      A     M      3.3;
      =     L      0.0;
      A     L      0.0;
      A     I     45.0;
      AN    I     45.1;
      =     M    612.2;
      A     L      0.0;
      AN    I     45.0;
      A     I     45.1;
      =     M    612.3;
NETWORK
TITLE =GUN3 1ST SHIFT ADV/REV END (LH ONLY)

      A     M      3.3;
      =     L      0.0;
      A     L      0.0;
      A     I     45.2;
      AN    I     45.3;
      =     M    612.4;
      A     L      0.0;
      AN    I     45.2;
      A     I     45.3;
      =     M    612.5;
NETWORK
TITLE =GUN3 2ND SHIFT ADV/REV END (LH ONLY)

      A     M      3.3;
      =     L      0.0;
      A     L      0.0;
      A     I     45.4;
      AN    I     45.5;
      =     M    612.6;
      A     L      0.0;
      AN    I     45.4;
      A     I     45.5;
      =     M    612.7;
NETWORK
TITLE =ALL CLAMP ADV/REV END

      A     M      3.3;
      =     L      0.0;
      A     L      0.0;
      A     M    610.2;
      A     M    610.4;
      =     M    618.0;
      A     L      0.0;
      A     M    610.3;
      A     M    610.5;
      =     M    618.1;
NETWORK
TITLE =GUN ALL HOME POSI.
//G3 SHIFT= LH ONLY
      A     M    612.1;
      A     M    612.2;
      A     M    612.5;
      A     M    612.7;
      =     M    618.2;
NETWORK
TITLE =PIN ADV
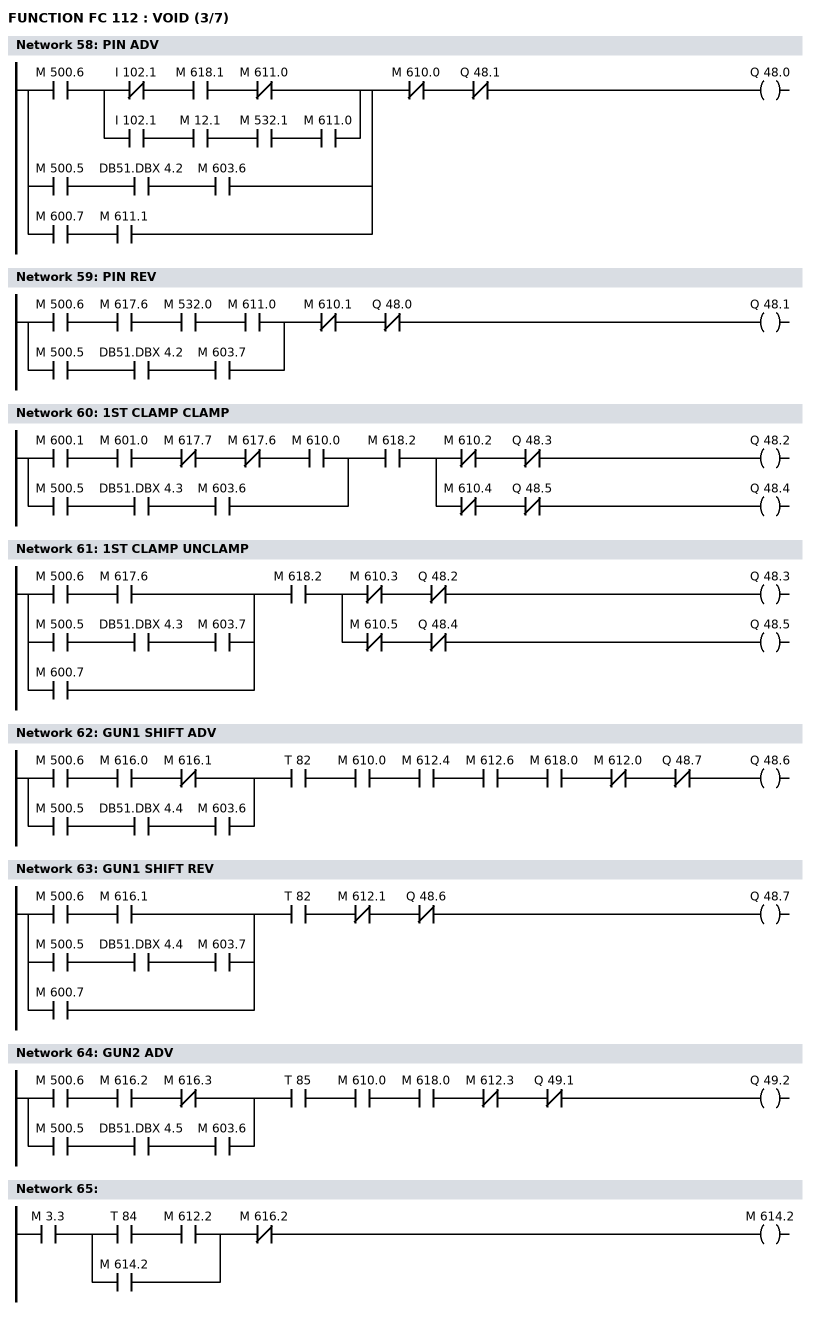

      A(    ;
      A     M    500.6;
      A(    ;
      AN    I    102.1;
      A     M    618.1;
      AN    M    611.0;
      O     ;
      A     I    102.1;
      A     M     12.1;
      A     M    532.1;
      A     M    611.0;
      )     ;
      O     ;
      A     M    500.5;
      A     DB51.DBX    4.2;
      A     M    603.6;
      O     ;
      A     M    600.7;
      A     M    611.1;
      )     ;
      AN    M    610.0;
      AN    Q     48.1;
      =     Q     48.0;
NETWORK
TITLE =PIN REV

      A(    ;
      A     M    500.6;
      A     M    617.6;
      A     M    532.0;
      A     M    611.0;
      O     ;
      A     M    500.5;
      A     DB51.DBX    4.2;
      A     M    603.7;
      )     ;
      AN    M    610.1;
      AN    Q     48.0;
      =     Q     48.1;
NETWORK
TITLE =1ST CLAMP CLAMP

      A(    ;
      A     M    600.1;
      A     M    601.0;
      AN    M    617.7;
      AN    M    617.6;
      A     M    610.0;
      O     ;
      A     M    500.5;
      A     DB51.DBX    4.3;
      A     M    603.6;
      )     ;
      A     M    618.2;
      =     L      0.0;
      A     L      0.0;
      AN    M    610.2;
      AN    Q     48.3;
      =     Q     48.2;
      A     L      0.0;
      AN    M    610.4;
      AN    Q     48.5;
      =     Q     48.4;
NETWORK
TITLE =1ST CLAMP UNCLAMP

      A(    ;
      A     M    500.6;
      A     M    617.6;
      O     ;
      A     M    500.5;
      A     DB51.DBX    4.3;
      A     M    603.7;
      O     M    600.7;
      )     ;
      A     M    618.2;
      =     L      0.0;
      A     L      0.0;
      AN    M    610.3;
      AN    Q     48.2;
      =     Q     48.3;
      A     L      0.0;
      AN    M    610.5;
      AN    Q     48.4;
      =     Q     48.5;
NETWORK
TITLE =GUN1 SHIFT ADV

      A(    ;
      A     M    500.6;
      A     M    616.0;
      AN    M    616.1;
      O     ;
      A     M    500.5;
      A     DB51.DBX    4.4;
      A     M    603.6;
      )     ;
      A     T     82;
      A     M    610.0;
      A     M    612.4;
      A     M    612.6;
      A     M    618.0;
      AN    M    612.0;
      AN    Q     48.7;
      =     Q     48.6;
NETWORK
TITLE =GUN1 SHIFT REV

      A(    ;
      A     M    500.6;
      A     M    616.1;
      O     ;
      A     M    500.5;
      A     DB51.DBX    4.4;
      A     M    603.7;
      O     M    600.7;
      )     ;
      A     T     82;
      AN    M    612.1;
      AN    Q     48.6;
      =     Q     48.7;
NETWORK
TITLE =GUN2 ADV

      A(    ;
      A     M    500.6;
      A     M    616.2;
      AN    M    616.3;
      O     ;
      A     M    500.5;
      A     DB51.DBX    4.5;
      A     M    603.6;
      )     ;
      A     T     85;
      A     M    610.0;
      A     M    618.0;
      AN    M    612.3;
      AN    Q     49.1;
      =     Q     49.2;
NETWORK
TITLE =

      A     M      3.3;
      A(    ;
      A     T     84;
      A     M    612.2;
      O     M    614.2;
      )     ;
      AN    M    616.2;
      =     M    614.2;
NETWORK
TITLE =GUN2 REV
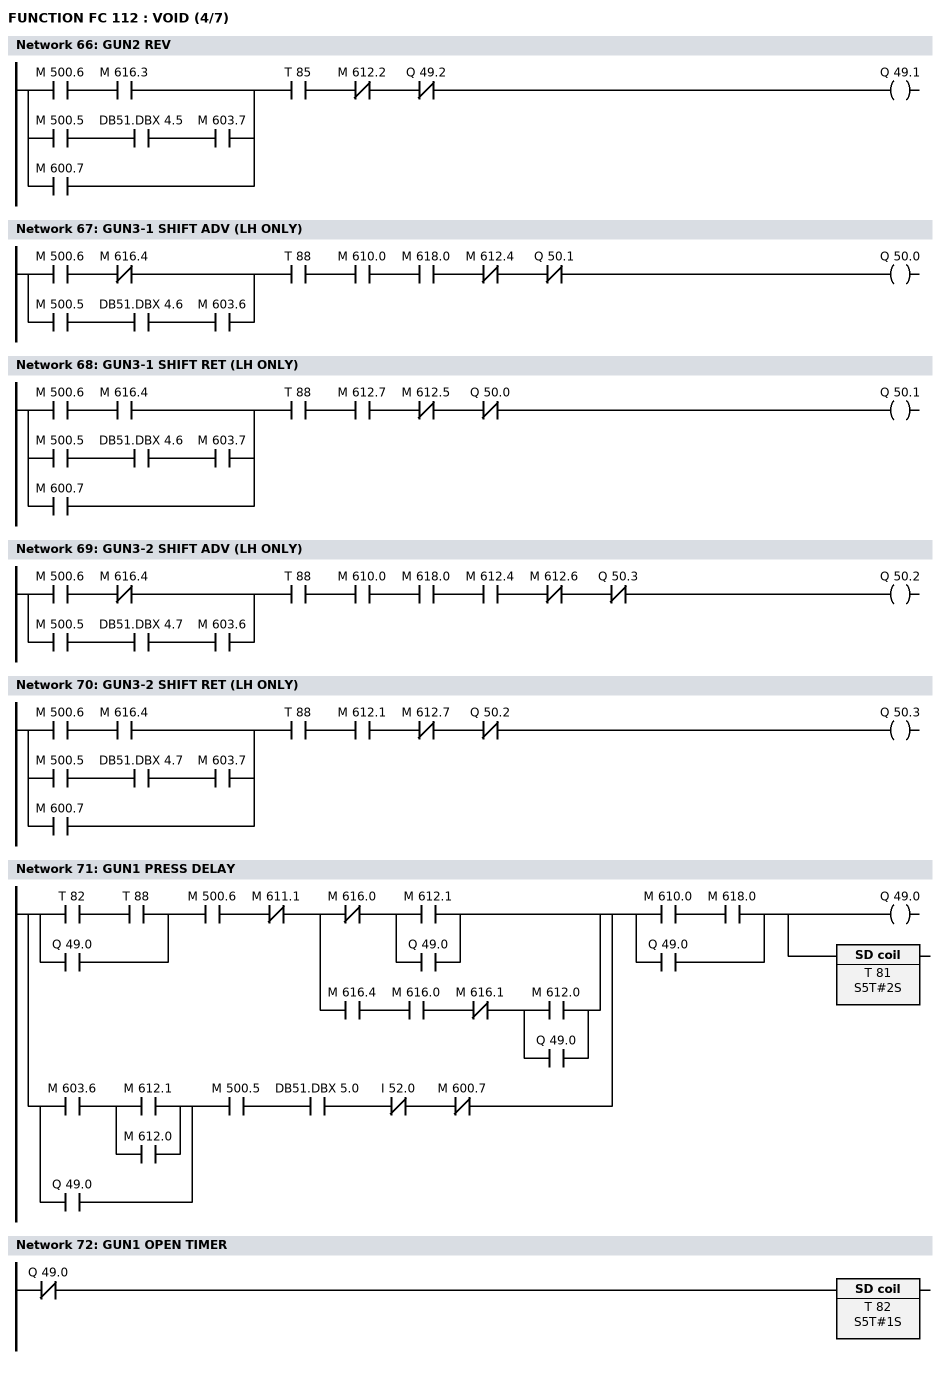

      A(    ;
      A     M    500.6;
      A     M    616.3;
      O     ;
      A     M    500.5;
      A     DB51.DBX    4.5;
      A     M    603.7;
      O     M    600.7;
      )     ;
      A     T     85;
      AN    M    612.2;
      AN    Q     49.2;
      =     Q     49.1;
NETWORK
TITLE =GUN3-1 SHIFT ADV (LH ONLY)

      A(    ;
      A     M    500.6;
      AN    M    616.4;
      O     ;
      A     M    500.5;
      A     DB51.DBX    4.6;
      A     M    603.6;
      )     ;
      A     T     88;
      A     M    610.0;
      A     M    618.0;
      AN    M    612.4;
      AN    Q     50.1;
      =     Q     50.0;
NETWORK
TITLE =GUN3-1 SHIFT RET (LH ONLY)

      A(    ;
      A     M    500.6;
      A     M    616.4;
      O     ;
      A     M    500.5;
      A     DB51.DBX    4.6;
      A     M    603.7;
      O     M    600.7;
      )     ;
      A     T     88;
      A     M    612.7;
      AN    M    612.5;
      AN    Q     50.0;
      =     Q     50.1;
NETWORK
TITLE =GUN3-2 SHIFT ADV (LH ONLY)

      A(    ;
      A     M    500.6;
      AN    M    616.4;
      O     ;
      A     M    500.5;
      A     DB51.DBX    4.7;
      A     M    603.6;
      )     ;
      A     T     88;
      A     M    610.0;
      A     M    618.0;
      A     M    612.4;
      AN    M    612.6;
      AN    Q     50.3;
      =     Q     50.2;
NETWORK
TITLE =GUN3-2 SHIFT RET (LH ONLY)

      A(    ;
      A     M    500.6;
      A     M    616.4;
      O     ;
      A     M    500.5;
      A     DB51.DBX    4.7;
      A     M    603.7;
      O     M    600.7;
      )     ;
      A     T     88;
      A     M    612.1;
      AN    M    612.7;
      AN    Q     50.2;
      =     Q     50.3;
NETWORK
TITLE =GUN1 PRESS DELAY

      A(    ;
      A(    ;
      A     T     82;
      A     T     88;
      O     Q     49.0;
      )     ;
      A     M    500.6;
      AN    M    611.1;
      A(    ;
      AN    M    616.0;
      A(    ;
      O     M    612.1;
      O     Q     49.0;
      )     ;
      O     ;
      A     M    616.4;
      A     M    616.0;
      AN    M    616.1;
      A(    ;
      O     M    612.0;
      O     Q     49.0;
      )     ;
      )     ;
      O     ;
      A(    ;
      A     M    603.6;
      A(    ;
      O     M    612.1;
      O     M    612.0;
      )     ;
      O     Q     49.0;
      )     ;
      A     M    500.5;
      A     DB51.DBX    5.0;
      AN    I     52.0;
      AN    M    600.7;
      )     ;
      A(    ;
      A     M    610.0;
      A     M    618.0;
      O     Q     49.0;
      )     ;
      =     Q     49.0;
      L     S5T#2S;
      SD    T     81;
NETWORK
TITLE =GUN1 OPEN TIMER

      AN    Q     49.0;
      L     S5T#1S;
      SD    T     82;
NETWORK
TITLE =GUN2 PRESS DELAY
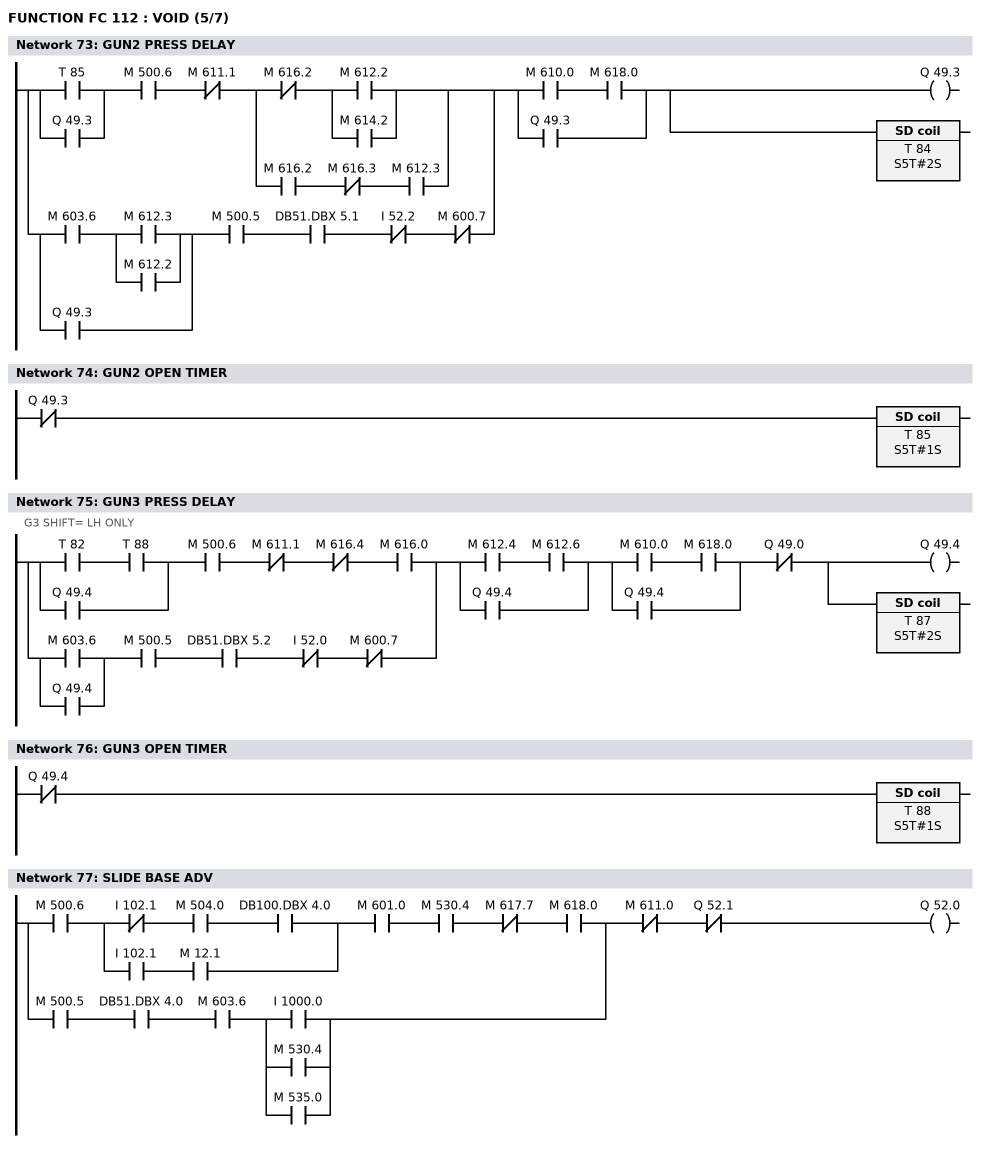

      A(    ;
      A(    ;
      O     T     85;
      O     Q     49.3;
      )     ;
      A     M    500.6;
      AN    M    611.1;
      A(    ;
      AN    M    616.2;
      A(    ;
      O     M    612.2;
      O     M    614.2;
      )     ;
      O     ;
      A     M    616.2;
      AN    M    616.3;
      A     M    612.3;
      )     ;
      O     ;
      A(    ;
      A     M    603.6;
      A(    ;
      O     M    612.3;
      O     M    612.2;
      )     ;
      O     Q     49.3;
      )     ;
      A     M    500.5;
      A     DB51.DBX    5.1;
      AN    I     52.2;
      AN    M    600.7;
      )     ;
      A(    ;
      A     M    610.0;
      A     M    618.0;
      O     Q     49.3;
      )     ;
      =     Q     49.3;
      L     S5T#2S;
      SD    T     84;
NETWORK
TITLE =GUN2 OPEN TIMER

      AN    Q     49.3;
      L     S5T#1S;
      SD    T     85;
NETWORK
TITLE =GUN3 PRESS DELAY
//G3 SHIFT= LH ONLY
      A(    ;
      A(    ;
      A     T     82;
      A     T     88;
      O     Q     49.4;
      )     ;
      A     M    500.6;
      AN    M    611.1;
      AN    M    616.4;
      A     M    616.0;
      O     ;
      A(    ;
      O     M    603.6;
      O     Q     49.4;
      )     ;
      A     M    500.5;
      A     DB51.DBX    5.2;
      AN    I     52.0;
      AN    M    600.7;
      )     ;
      A(    ;
      A     M    612.4;
      A     M    612.6;
      O     Q     49.4;
      )     ;
      A(    ;
      A     M    610.0;
      A     M    618.0;
      O     Q     49.4;
      )     ;
      AN    Q     49.0;
      =     Q     49.4;
      L     S5T#2S;
      SD    T     87;
NETWORK
TITLE =GUN3 OPEN TIMER

      AN    Q     49.4;
      L     S5T#1S;
      SD    T     88;
NETWORK
TITLE =SLIDE BASE ADV

      A(    ;
      A     M    500.6;
      A(    ;
      AN    I    102.1;
      A     M    504.0;
      A     DB100.DBX    4.0;
      O     ;
      A     I    102.1;
      A     M     12.1;
      )     ;
      A     M    601.0;
      A     M    530.4;
      AN    M    617.7;
      A     M    618.0;
      O     ;
      A     M    500.5;
      A     DB51.DBX    4.0;
      A     M    603.6;
      A(    ;
      O     I   1000.0;
      O     M    530.4;
      O     M    535.0;
      )     ;
      )     ;
      AN    M    611.0;
      AN    Q     52.1;
      =     Q     52.0;
NETWORK
TITLE =SLIDE BASE REV
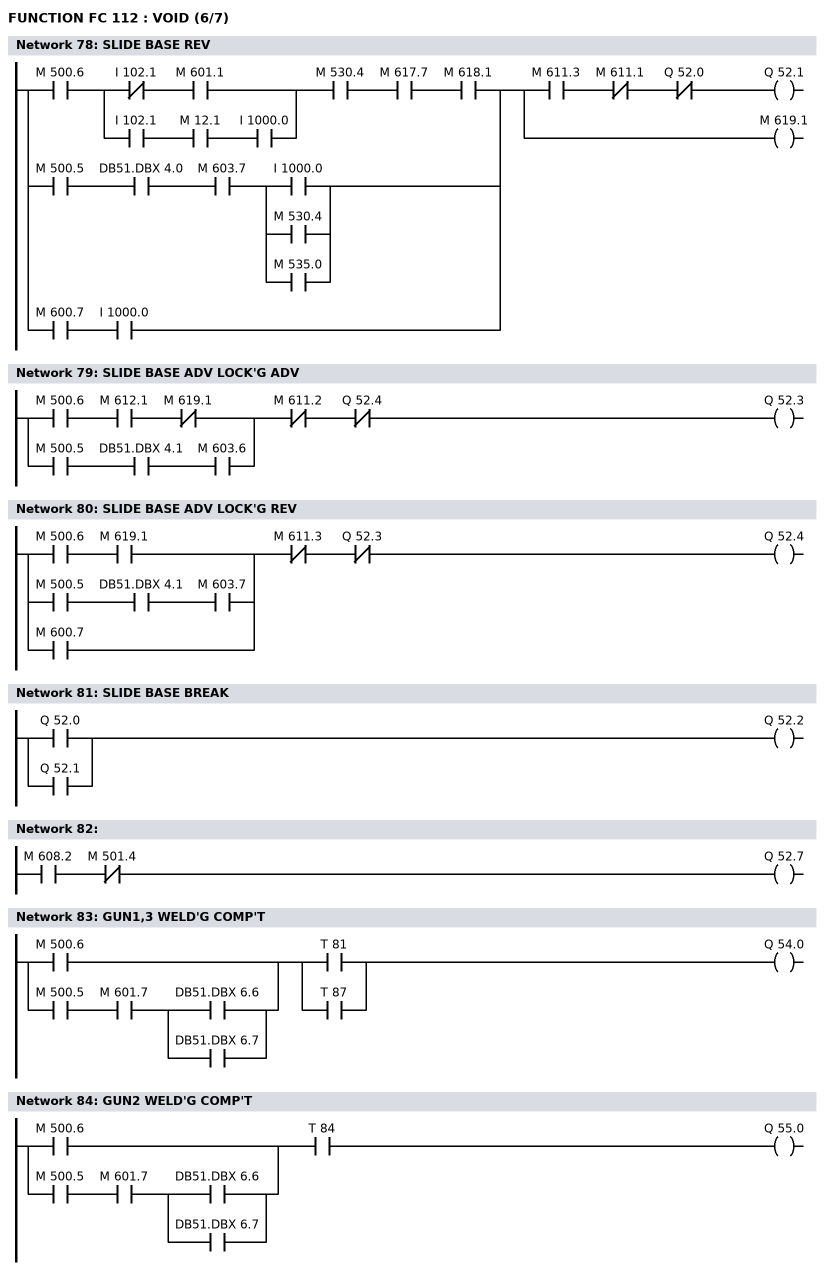

      A     M    500.6;
      A(    ;
      AN    I    102.1;
      A     M    601.1;
      O     ;
      A     I    102.1;
      A     M     12.1;
      A     I   1000.0;
      )     ;
      A     M    530.4;
      A     M    617.7;
      A     M    618.1;
      O     ;
      A     M    500.5;
      A     DB51.DBX    4.0;
      A     M    603.7;
      A(    ;
      O     I   1000.0;
      O     M    530.4;
      O     M    535.0;
      )     ;
      O     ;
      A     M    600.7;
      A     I   1000.0;
      =     L      0.0;
      A     L      0.0;
      A     M    611.3;
      AN    M    611.1;
      AN    Q     52.0;
      =     Q     52.1;
      A     L      0.0;
      BLD   102;
      =     M    619.1;
NETWORK
TITLE =SLIDE BASE ADV LOCK'G ADV

      A(    ;
      A     M    500.6;
      A     M    612.1;
      AN    M    619.1;
      O     ;
      A     M    500.5;
      A     DB51.DBX    4.1;
      A     M    603.6;
      )     ;
      AN    M    611.2;
      AN    Q     52.4;
      =     Q     52.3;
NETWORK
TITLE =SLIDE BASE ADV LOCK'G REV

      A(    ;
      A     M    500.6;
      A     M    619.1;
      O     ;
      A     M    500.5;
      A     DB51.DBX    4.1;
      A     M    603.7;
      O     M    600.7;
      )     ;
      AN    M    611.3;
      AN    Q     52.3;
      =     Q     52.4;
NETWORK
TITLE =SLIDE BASE BREAK

      O     Q     52.0;
      O     Q     52.1;
      =     Q     52.2;
NETWORK
TITLE =

      A     M    608.2;
      AN    M    501.4;
      =     Q     52.7;
NETWORK
TITLE =GUN1,3 WELD'G COMP'T

      A(    ;
      O     M    500.6;
      O     ;
      A     M    500.5;
      A     M    601.7;
      A(    ;
      O     DB51.DBX    6.6;
      O     DB51.DBX    6.7;
      )     ;
      )     ;
      A(    ;
      O     T     81;
      O     T     87;
      )     ;
      =     Q     54.0;
NETWORK
TITLE =GUN2 WELD'G COMP'T

      A(    ;
      O     M    500.6;
      O     ;
      A     M    500.5;
      A     M    601.7;
      A(    ;
      O     DB51.DBX    6.6;
      O     DB51.DBX    6.7;
      )     ;
      )     ;
      A     T     84;
      =     Q     55.0;
NETWORK
TITLE =GUN1,3 WELD'G TEST
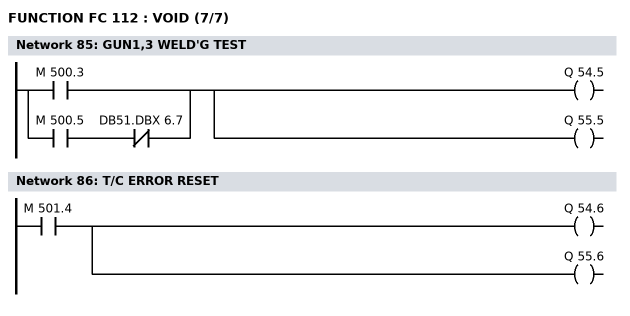

      O     M    500.3;
      O     ;
      A     M    500.5;
      AN    DB51.DBX    6.7;
      =     Q     54.5;
      =     Q     55.5;
NETWORK
TITLE =T/C ERROR RESET

      A     M    501.4;
      =     Q     54.6;
      =     Q     55.6;
END_FUNCTION

FUNCTION FC 113 : VOID
TITLE =
VERSION : 0.1

BEGIN
NETWORK
TITLE =BODY NO.
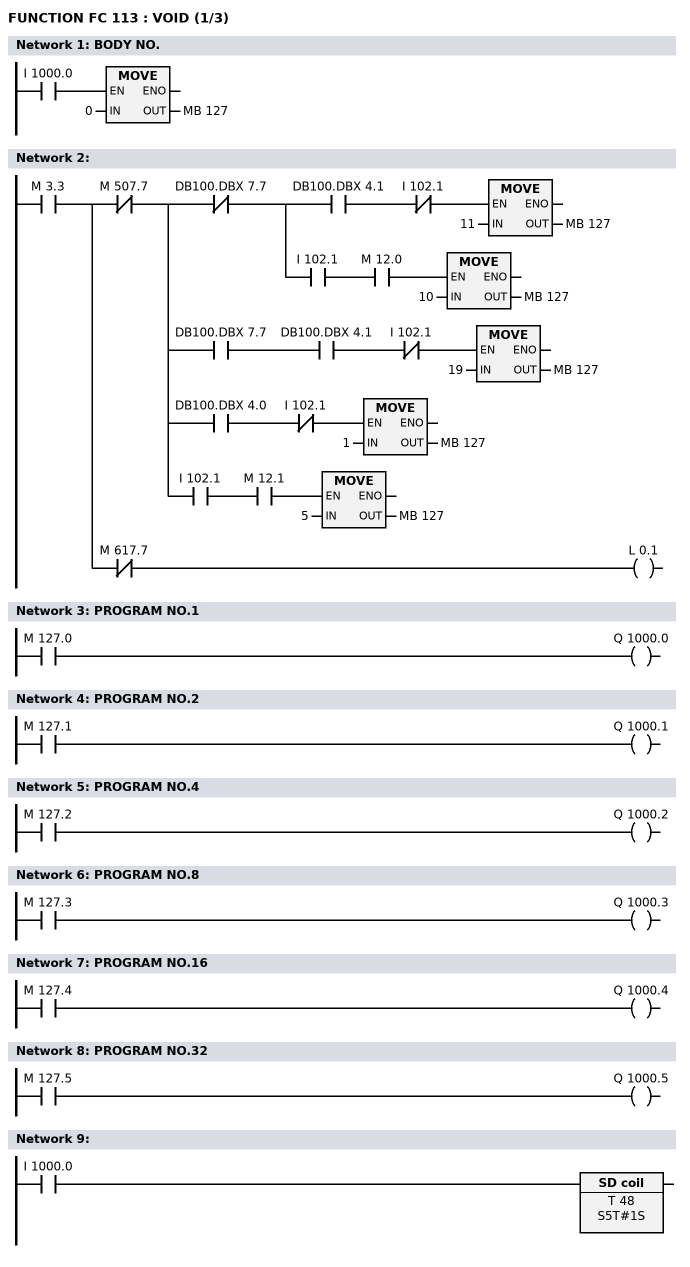

      A     I   1000.0;
      JNB   _001;
      L     0;
      T     MB   127;
_001: NOP   0;
NETWORK
TITLE =

      A     M      3.3;
      =     L      0.0;
      A     L      0.0;
      AN    M    507.7;
      =     L      0.1;
      A     L      0.1;
      AN    DB100.DBX    7.7;
      =     L      0.2;
      A     L      0.2;
      A     DB100.DBX    4.1;
      AN    I    102.1;
      JNB   _002;
      L     11;
      T     MB   127;
_002: NOP   0;
      A     L      0.2;
      A     I    102.1;
      A     M     12.0;
      JNB   _003;
      L     10;
      T     MB   127;
_003: NOP   0;
      A     L      0.1;
      A     DB100.DBX    7.7;
      A     DB100.DBX    4.1;
      AN    I    102.1;
      JNB   _004;
      L     19;
      T     MB   127;
_004: NOP   0;
      A     L      0.0;
      AN    M    617.7;
      =     L      0.1;
      A     L      0.1;
      A     DB100.DBX    4.0;
      AN    I    102.1;
      JNB   _005;
      L     1;
      T     MB   127;
_005: NOP   0;
      A     L      0.1;
      A     I    102.1;
      A     M     12.1;
      JNB   _006;
      L     5;
      T     MB   127;
_006: NOP   0;
NETWORK
TITLE =PROGRAM NO.1

      A     M    127.0;
      =     Q   1000.0;
NETWORK
TITLE =PROGRAM NO.2

      A     M    127.1;
      =     Q   1000.1;
NETWORK
TITLE =PROGRAM NO.4

      A     M    127.2;
      =     Q   1000.2;
NETWORK
TITLE =PROGRAM NO.8

      A     M    127.3;
      =     Q   1000.3;
NETWORK
TITLE =PROGRAM NO.16

      A     M    127.4;
      =     Q   1000.4;
NETWORK
TITLE =PROGRAM NO.32

      A     M    127.5;
      =     Q   1000.5;
NETWORK
TITLE =

      A     I   1000.0;
      L     S5T#1S;
      SD    T     48;
NETWORK
TITLE =
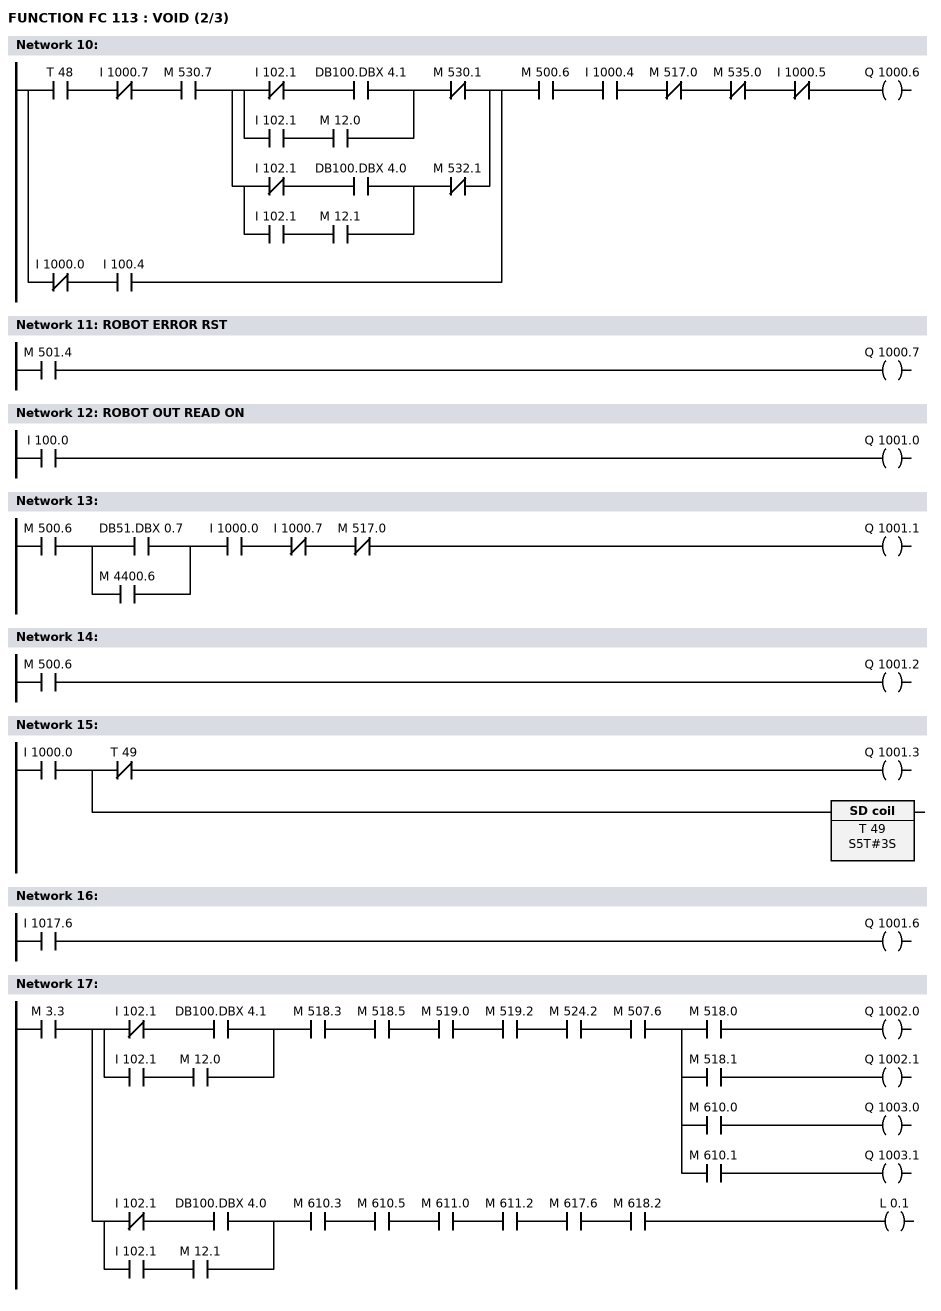

      A(    ;
      A     T     48;
      AN    I   1000.7;
      A     M    530.7;
      A(    ;
      A(    ;
      AN    I    102.1;
      A     DB100.DBX    4.1;
      O     ;
      A     I    102.1;
      A     M     12.0;
      )     ;
      AN    M    530.1;
      O     ;
      A(    ;
      AN    I    102.1;
      A     DB100.DBX    4.0;
      O     ;
      A     I    102.1;
      A     M     12.1;
      )     ;
      AN    M    532.1;
      )     ;
      O     ;
      AN    I   1000.0;
      A     I    100.4;
      )     ;
      A     M    500.6;
      A     I   1000.4;
      AN    M    517.0;
      AN    M    535.0;
      AN    I   1000.5;
      =     Q   1000.6;
NETWORK
TITLE =ROBOT ERROR RST

      A     M    501.4;
      =     Q   1000.7;
NETWORK
TITLE =ROBOT OUT READ ON

      A     I    100.0;
      =     Q   1001.0;
NETWORK
TITLE =

      A     M    500.6;
      A(    ;
      O     DB51.DBX    0.7;
      O     M   4400.6;
      )     ;
      A     I   1000.0;
      AN    I   1000.7;
      AN    M    517.0;
      =     Q   1001.1;
NETWORK
TITLE =

      A     M    500.6;
      =     Q   1001.2;
NETWORK
TITLE =

      A     I   1000.0;
      =     L      0.0;
      A     L      0.0;
      AN    T     49;
      =     Q   1001.3;
      A     L      0.0;
      BLD   102;
      L     S5T#3S;
      SD    T     49;
NETWORK
TITLE =

      A     I   1017.6;
      =     Q   1001.6;
NETWORK
TITLE =

      A     M      3.3;
      =     L      0.0;
      A     L      0.0;
      A(    ;
      AN    I    102.1;
      A     DB100.DBX    4.1;
      O     ;
      A     I    102.1;
      A     M     12.0;
      )     ;
      A     M    518.3;
      A     M    518.5;
      A     M    519.0;
      A     M    519.2;
      A     M    524.2;
      A     M    507.6;
      =     L      0.1;
      A     L      0.1;
      A     M    518.0;
      =     Q   1002.0;
      A     L      0.1;
      A     M    518.1;
      =     Q   1002.1;
      A     L      0.0;
      A(    ;
      AN    I    102.1;
      A     DB100.DBX    4.0;
      O     ;
      A     I    102.1;
      A     M     12.1;
      )     ;
      A     M    610.3;
      A     M    610.5;
      A     M    611.0;
      A     M    611.2;
      A     M    617.6;
      A     M    618.2;
      =     L      0.1;
      A     L      0.1;
      A     M    610.0;
      =     Q   1003.0;
      A     L      0.1;
      A     M    610.1;
      =     Q   1003.1;
NETWORK
TITLE =
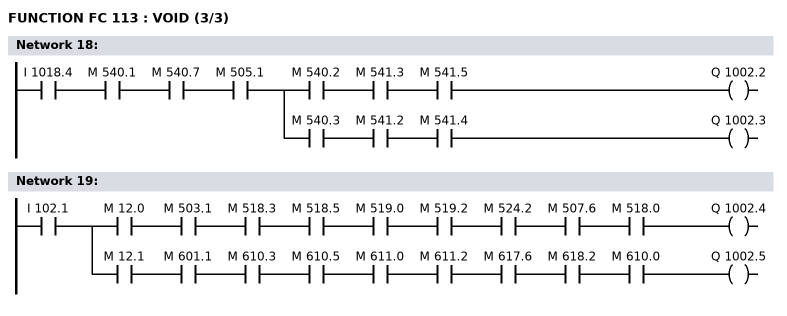

      A     I   1018.4;
      A     M    540.1;
      A     M    540.7;
      A     M    505.1;
      =     L      0.0;
      A     L      0.0;
      A     M    540.2;
      A     M    541.3;
      A     M    541.5;
      =     Q   1002.2;
      A     L      0.0;
      A     M    540.3;
      A     M    541.2;
      A     M    541.4;
      =     Q   1002.3;
NETWORK
TITLE =

      A     I    102.1;
      =     L      0.0;
      A     L      0.0;
      A     M     12.0;
      A     M    503.1;
      A     M    518.3;
      A     M    518.5;
      A     M    519.0;
      A     M    519.2;
      A     M    524.2;
      A     M    507.6;
      A     M    518.0;
      =     Q   1002.4;
      A     L      0.0;
      A     M     12.1;
      A     M    601.1;
      A     M    610.3;
      A     M    610.5;
      A     M    611.0;
      A     M    611.2;
      A     M    617.6;
      A     M    618.2;
      A     M    610.0;
      =     Q   1002.5;
END_FUNCTION

FUNCTION_BLOCK FB 120
TITLE =
VERSION : 0.1


VAR
  S711_MODE : FB 402;
END_VAR
BEGIN
NETWORK
TITLE =
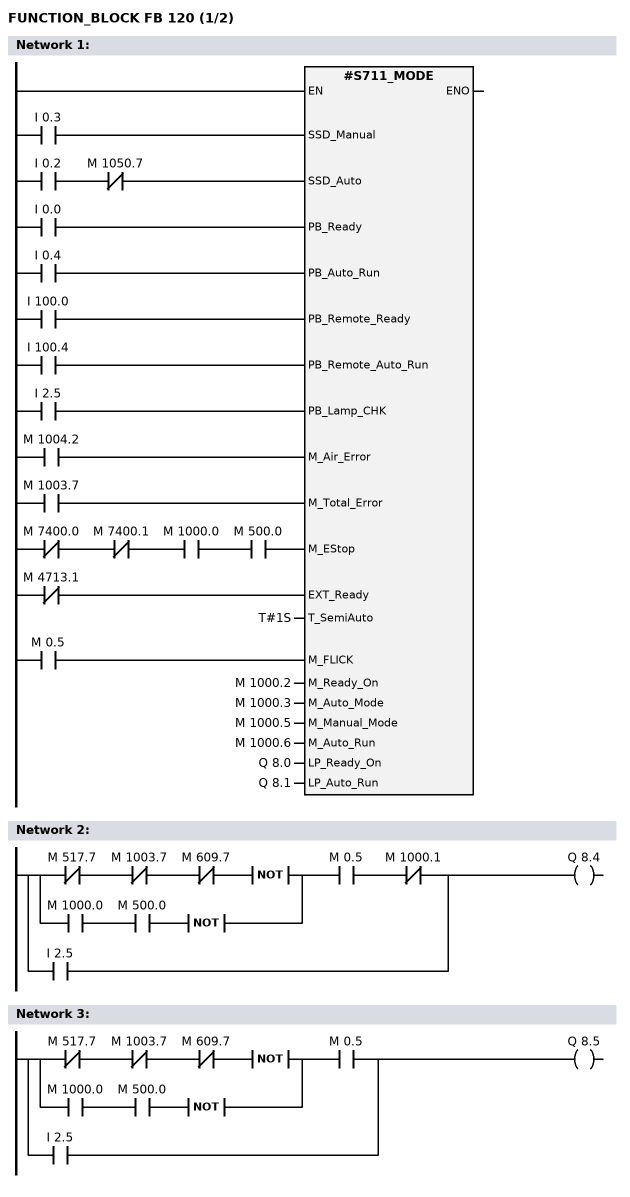

      A     I      0.3;
      =     L      0.0;
      BLD   103;
      A     I      0.2;
      AN    M   1050.7;
      =     L      0.1;
      BLD   103;
      A     I      0.0;
      =     L      0.2;
      BLD   103;
      A     I      0.4;
      =     L      0.3;
      BLD   103;
      A     I    100.0;
      =     L      0.4;
      BLD   103;
      A     I    100.4;
      =     L      0.5;
      BLD   103;
      A     I      2.5;
      =     L      0.6;
      BLD   103;
      A     M   1004.2;
      =     L      0.7;
      BLD   103;
      A     M   1003.7;
      =     L      1.1;
      BLD   103;
      AN    M   7400.0;
      AN    M   7400.1;
      A     M   1000.0;
      A     M    500.0;
      =     L      1.2;
      BLD   103;
      AN    M   4713.1;
      =     L      1.3;
      BLD   103;
      A     M      0.5;
      =     L      1.5;
      BLD   103;
      CALL #S711_MODE (
           SSD_Manual               := L      0.0,
           SSD_Auto                 := L      0.1,
           PB_Ready                 := L      0.2,
           PB_Auto_Run              := L      0.3,
           PB_Remote_Ready          := L      0.4,
           PB_Remote_Auto_Run       := L      0.5,
           PB_Lamp_CHK              := L      0.6,
           M_Air_Error              := L      0.7,
           M_Total_Error            := L      1.1,
           M_EStop                  := L      1.2,
           EXT_Ready                := L      1.3,
           T_SemiAuto               := T#1S,
           M_FLICK                  := L      1.5,
           M_Ready_On               := M   1000.2,
           M_Auto_Mode              := M   1000.3,
           M_Manual_Mode            := M   1000.5,
           M_Auto_Run               := M   1000.6,
           LP_Ready_On              := Q      8.0,
           LP_Auto_Run              := Q      8.1);
      NOP   0;
NETWORK
TITLE =

      A(    ;
      AN    M    517.7;
      AN    M   1003.7;
      AN    M    609.7;
      NOT   ;
      O(    ;
      A     M   1000.0;
      A     M    500.0;
      NOT   ;
      )     ;
      )     ;
      A     M      0.5;
      AN    M   1000.1;
      O     I      2.5;
      =     Q      8.4;
NETWORK
TITLE =

      A(    ;
      AN    M    517.7;
      AN    M   1003.7;
      AN    M    609.7;
      NOT   ;
      O(    ;
      A     M   1000.0;
      A     M    500.0;
      NOT   ;
      )     ;
      )     ;
      A     M      0.5;
      O     I      2.5;
      =     Q      8.5;
NETWORK
TITLE =
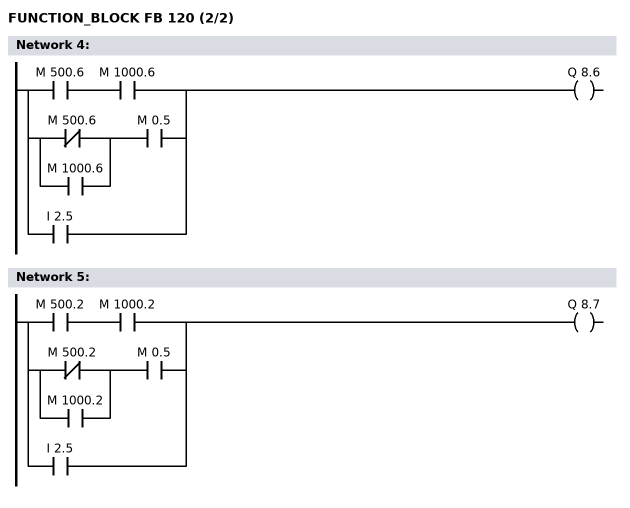

      A     M    500.6;
      A     M   1000.6;
      O     ;
      A(    ;
      ON    M    500.6;
      O     M   1000.6;
      )     ;
      A     M      0.5;
      O     I      2.5;
      =     Q      8.6;
NETWORK
TITLE =

      A     M    500.2;
      A     M   1000.2;
      O     ;
      A(    ;
      ON    M    500.2;
      O     M   1000.2;
      )     ;
      A     M      0.5;
      O     I      2.5;
      =     Q      8.7;
END_FUNCTION_BLOCK

DATA_BLOCK DB 120
TITLE =
VERSION : 0.0

 FB 120
BEGIN
   S711_MODE.SSD_Manual := FALSE;
   S711_MODE.SSD_Auto := FALSE;
   S711_MODE.PB_Ready := FALSE;
   S711_MODE.PB_Auto_Run := FALSE;
   S711_MODE.PB_Remote_Ready := FALSE;
   S711_MODE.PB_Remote_Auto_Run := FALSE;
   S711_MODE.PB_Lamp_CHK := FALSE;
   S711_MODE.M_Air_Error := FALSE;
   S711_MODE.M_Water_Error := FALSE;
   S711_MODE.M_Total_Error := FALSE;
   S711_MODE.M_EStop := FALSE;
   S711_MODE.EXT_Ready := FALSE;
   S711_MODE.EXT_Auto := FALSE;
   S711_MODE.T_SemiAuto := T#0MS;
   S711_MODE.M_FLICK := FALSE;
   S711_MODE.M_Ready_On := FALSE;
   S711_MODE.M_Auto_Mode := FALSE;
   S711_MODE.M_SemiAuto_Mode := FALSE;
   S711_MODE.M_Manual_Mode := FALSE;
   S711_MODE.M_Auto_Run := FALSE;
   S711_MODE.LP_Ready_On := FALSE;
   S711_MODE.LP_Auto_Run := FALSE;
   S711_MODE.AUTO_MODE_DELAY.IN := FALSE;
   S711_MODE.AUTO_MODE_DELAY.PT := T#0MS;
   S711_MODE.AUTO_MODE_DELAY.Q := FALSE;
   S711_MODE.AUTO_MODE_DELAY.ET := T#0MS;
   S711_MODE.AUTO_MODE_DELAY.STATE := B#16#0;
   S711_MODE.AUTO_MODE_DELAY.STIME := T#0MS;
   S711_MODE.AUTO_MODE_DELAY.ATIME := T#0MS;
   S711_MODE.SEMI_AUTO_DELAY.IN := FALSE;
   S711_MODE.SEMI_AUTO_DELAY.PT := T#0MS;
   S711_MODE.SEMI_AUTO_DELAY.Q := FALSE;
   S711_MODE.SEMI_AUTO_DELAY.ET := T#0MS;
   S711_MODE.SEMI_AUTO_DELAY.STATE := B#16#0;
   S711_MODE.SEMI_AUTO_DELAY.STIME := T#0MS;
   S711_MODE.SEMI_AUTO_DELAY.ATIME := T#0MS;
   S711_MODE.MANUAL_DELAY.IN := FALSE;
   S711_MODE.MANUAL_DELAY.PT := T#0MS;
   S711_MODE.MANUAL_DELAY.Q := FALSE;
   S711_MODE.MANUAL_DELAY.ET := T#0MS;
   S711_MODE.MANUAL_DELAY.STATE := B#16#0;
   S711_MODE.MANUAL_DELAY.STIME := T#0MS;
   S711_MODE.MANUAL_DELAY.ATIME := T#0MS;
END_DATA_BLOCK

FUNCTION FC 120 : VOID
TITLE =
VERSION : 0.1

BEGIN
NETWORK
TITLE =
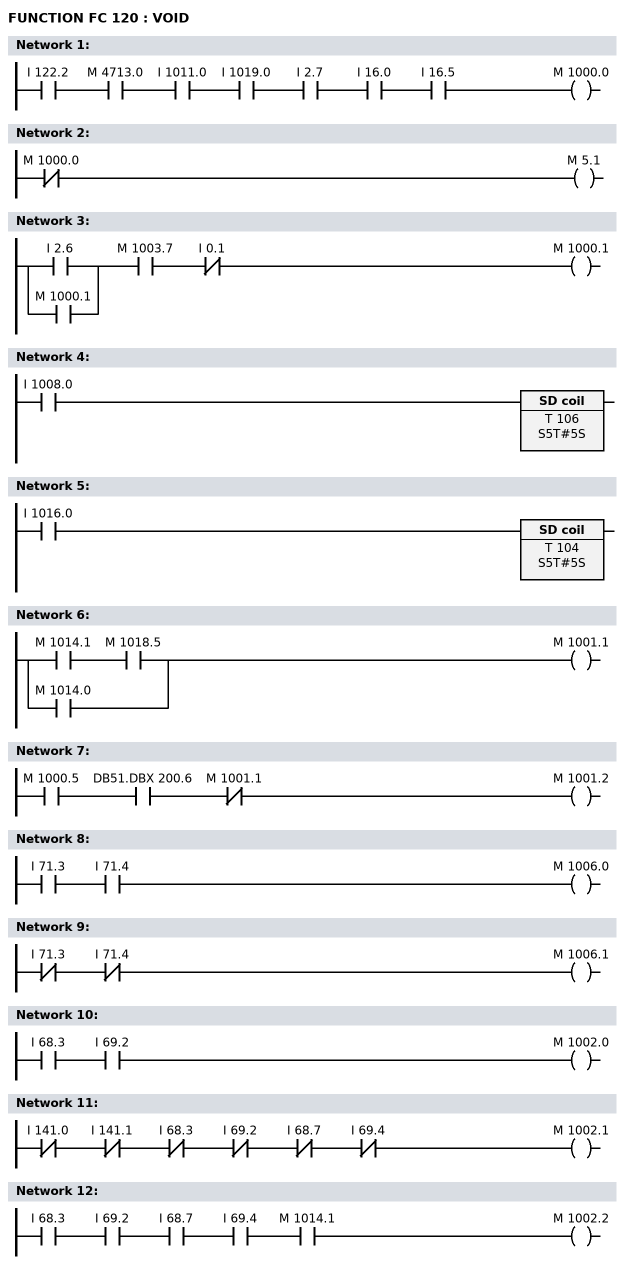

      A     I    122.2;
      A     M   4713.0;
      A     I   1011.0;
      A     I   1019.0;
      A     I      2.7;
      A     I     16.0;
      A     I     16.5;
      =     M   1000.0;
NETWORK
TITLE =

      AN    M   1000.0;
      =     M      5.1;
NETWORK
TITLE =

      A(    ;
      O     I      2.6;
      O     M   1000.1;
      )     ;
      A     M   1003.7;
      AN    I      0.1;
      =     M   1000.1;
NETWORK
TITLE =

      A     I   1008.0;
      L     S5T#5S;
      SD    T    106;
NETWORK
TITLE =

      A     I   1016.0;
      L     S5T#5S;
      SD    T    104;
NETWORK
TITLE =

      A     M   1014.1;
      A     M   1018.5;
      O     M   1014.0;
      =     M   1001.1;
NETWORK
TITLE =

      A     M   1000.5;
      A     DB51.DBX  200.6;
      AN    M   1001.1;
      =     M   1001.2;
NETWORK
TITLE =

      A     I     71.3;
      A     I     71.4;
      =     M   1006.0;
NETWORK
TITLE =

      AN    I     71.3;
      AN    I     71.4;
      =     M   1006.1;
NETWORK
TITLE =

      A     I     68.3;
      A     I     69.2;
      =     M   1002.0;
NETWORK
TITLE =

      AN    I    141.0;
      AN    I    141.1;
      AN    I     68.3;
      AN    I     69.2;
      AN    I     68.7;
      AN    I     69.4;
      =     M   1002.1;
NETWORK
TITLE =

      A     I     68.3;
      A     I     69.2;
      A     I     68.7;
      A     I     69.4;
      A     M   1014.1;
      =     M   1002.2;
NETWORK
TITLE =

      AN    OV;
      =     L      0.0;
      A     L      0.0;
      A     I     68.3;
      A     I     69.2;
      A     I     68.7;
      A     I     69.4;
      =     M   1019.0;
      A     L      0.0;
      AN    I    141.0;
      AN    I    141.1;
      AN    I     68.3;
      AN    I     69.2;
      AN    I     68.7;
      AN    I     69.4;
      =     M   1019.1;
NETWORK
TITLE =
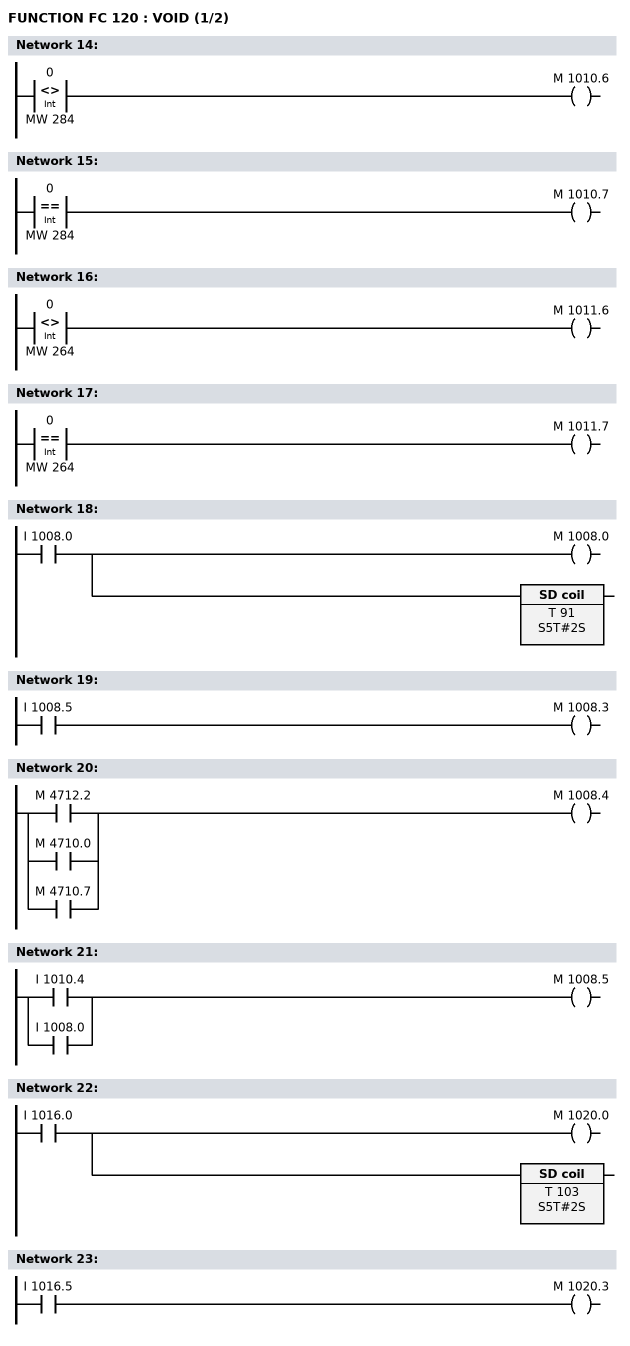

      L     0;
      L     MW   284;
      <>I   ;
      =     M   1010.6;
NETWORK
TITLE =

      L     0;
      L     MW   284;
      ==I   ;
      =     M   1010.7;
NETWORK
TITLE =

      L     0;
      L     MW   264;
      <>I   ;
      =     M   1011.6;
NETWORK
TITLE =

      L     0;
      L     MW   264;
      ==I   ;
      =     M   1011.7;
NETWORK
TITLE =

      A     I   1008.0;
      =     M   1008.0;
      L     S5T#2S;
      SD    T     91;
NETWORK
TITLE =

      A     I   1008.5;
      =     M   1008.3;
NETWORK
TITLE =

      O     M   4712.2;
      O     M   4710.0;
      O     M   4710.7;
      =     M   1008.4;
NETWORK
TITLE =

      O     I   1010.4;
      O     I   1008.0;
      =     M   1008.5;
NETWORK
TITLE =

      A     I   1016.0;
      =     M   1020.0;
      L     S5T#2S;
      SD    T    103;
NETWORK
TITLE =

      A     I   1016.5;
      =     M   1020.3;
NETWORK
TITLE =
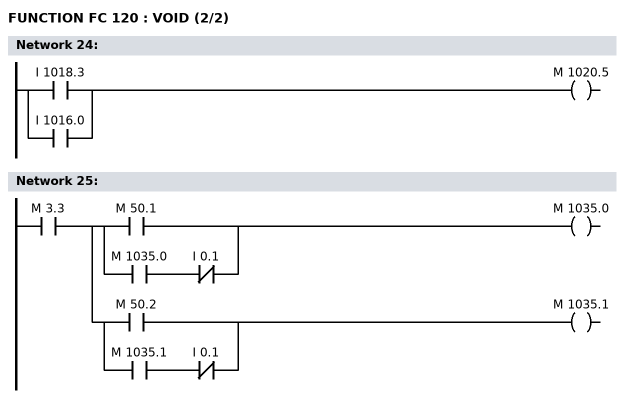

      O     I   1018.3;
      O     I   1016.0;
      =     M   1020.5;
NETWORK
TITLE =

      A     M      3.3;
      =     L      0.0;
      A     L      0.0;
      A(    ;
      O     M     50.1;
      O     ;
      A     M   1035.0;
      AN    I      0.1;
      )     ;
      =     M   1035.0;
      A     L      0.0;
      A(    ;
      O     M     50.2;
      O     ;
      A     M   1035.1;
      AN    I      0.1;
      )     ;
      =     M   1035.1;
END_FUNCTION

FUNCTION_BLOCK FB 121
TITLE =
VERSION : 0.1


VAR
  INDEX_LOCK : FB 424;
  TL_BT_CHANGE : FB 424;
  TL_PIN : FB 424;
  LM_BT_CHANGE : FB 430;
  LM_CLAMP : FB 424;
  LM_PIN : FB 424;
  LM_INDEX_CLAMP : FB 424;
  LM_INDEX_PIN : FB 424;
  INR_PLT3_UP_DOWN : FB 424;
  INR_PLT3_LOCK : FB 424;
  INR_PLT4_UP_DOWN : FB 424;
  INR_PLT4_LOCK : FB 424;
  INR_PLT5_UP_DOWN : FB 424;
  INR_PLT5_LOCK : FB 424;
END_VAR
BEGIN
NETWORK
TITLE =#711 COMPL LS이상

NETWORK
TITLE =
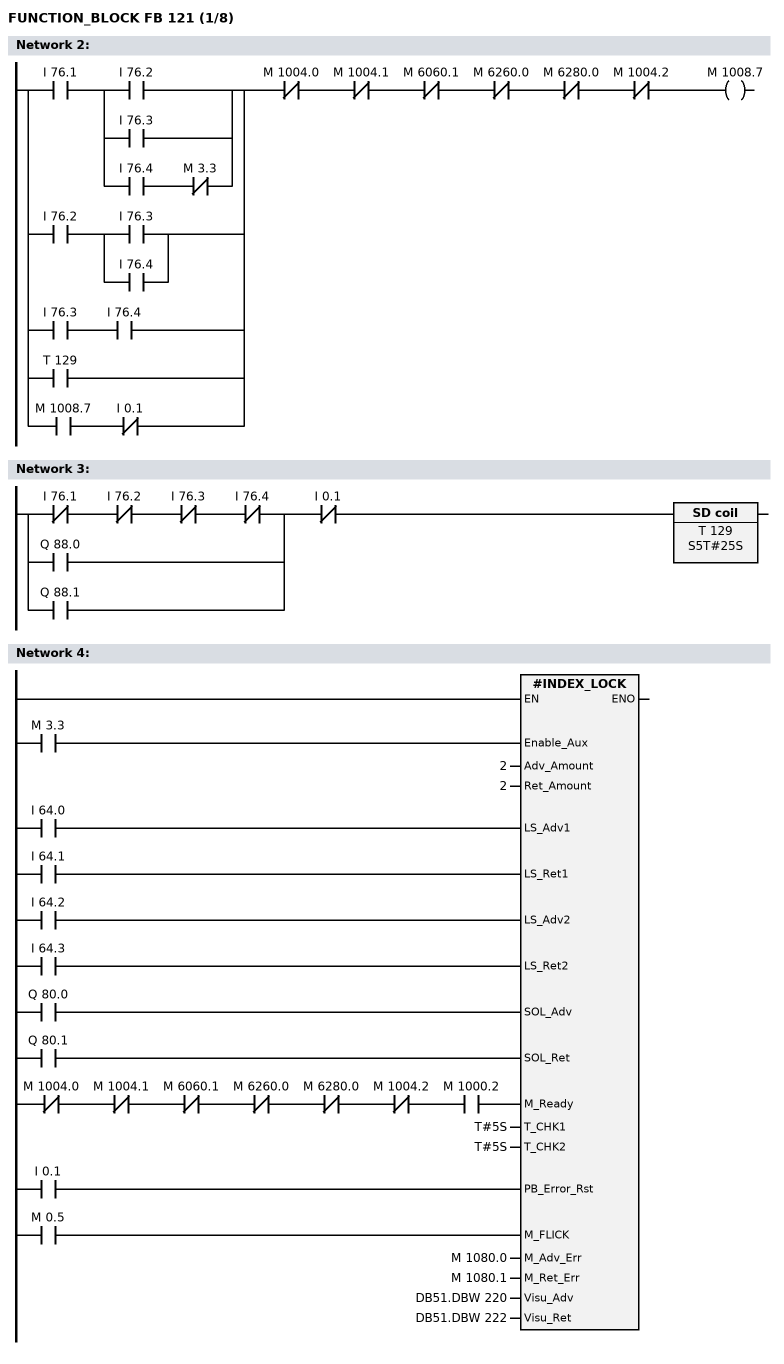

      A(    ;
      A     I     76.1;
      A(    ;
      O     I     76.2;
      O     I     76.3;
      O     ;
      A     I     76.4;
      AN    M      3.3;
      )     ;
      O     ;
      A     I     76.2;
      A(    ;
      O     I     76.3;
      O     I     76.4;
      )     ;
      O     ;
      A     I     76.3;
      A     I     76.4;
      O     T    129;
      O     ;
      A     M   1008.7;
      AN    I      0.1;
      )     ;
      AN    M   1004.0;
      AN    M   1004.1;
      AN    M   6060.1;
      AN    M   6260.0;
      AN    M   6280.0;
      AN    M   1004.2;
      =     M   1008.7;
NETWORK
TITLE =

      A(    ;
      AN    I     76.1;
      AN    I     76.2;
      AN    I     76.3;
      AN    I     76.4;
      O     Q     88.0;
      O     Q     88.1;
      )     ;
      AN    I      0.1;
      L     S5T#25S;
      SD    T    129;
NETWORK
TITLE =

      A     M      3.3;
      =     L      0.0;
      BLD   103;
      A     I     64.0;
      =     L      0.1;
      BLD   103;
      A     I     64.1;
      =     L      0.2;
      BLD   103;
      A     I     64.2;
      =     L      0.3;
      BLD   103;
      A     I     64.3;
      =     L      0.4;
      BLD   103;
      A     Q     80.0;
      =     L      1.1;
      BLD   103;
      A     Q     80.1;
      =     L      1.2;
      BLD   103;
      AN    M   1004.0;
      AN    M   1004.1;
      AN    M   6060.1;
      AN    M   6260.0;
      AN    M   6280.0;
      AN    M   1004.2;
      A     M   1000.2;
      =     L      1.3;
      BLD   103;
      A     I      0.1;
      =     L      1.5;
      BLD   103;
      A     M      0.5;
      =     L      1.6;
      BLD   103;
      CALL #INDEX_LOCK (
           Enable_Aux               := L      0.0,
           Adv_Amount               := 2,
           Ret_Amount               := 2,
           LS_Adv1                  := L      0.1,
           LS_Ret1                  := L      0.2,
           LS_Adv2                  := L      0.3,
           LS_Ret2                  := L      0.4,
           SOL_Adv                  := L      1.1,
           SOL_Ret                  := L      1.2,
           M_Ready                  := L      1.3,
           T_CHK1                   := T#5S,
           T_CHK2                   := T#5S,
           PB_Error_Rst             := L      1.5,
           M_FLICK                  := L      1.6,
           M_Adv_Err                := M   1080.0,
           M_Ret_Err                := M   1080.1,
           Visu_Adv                 := DB51.DBW  220,
           Visu_Ret                 := DB51.DBW  222);
      NOP   0;
NETWORK
TITLE =
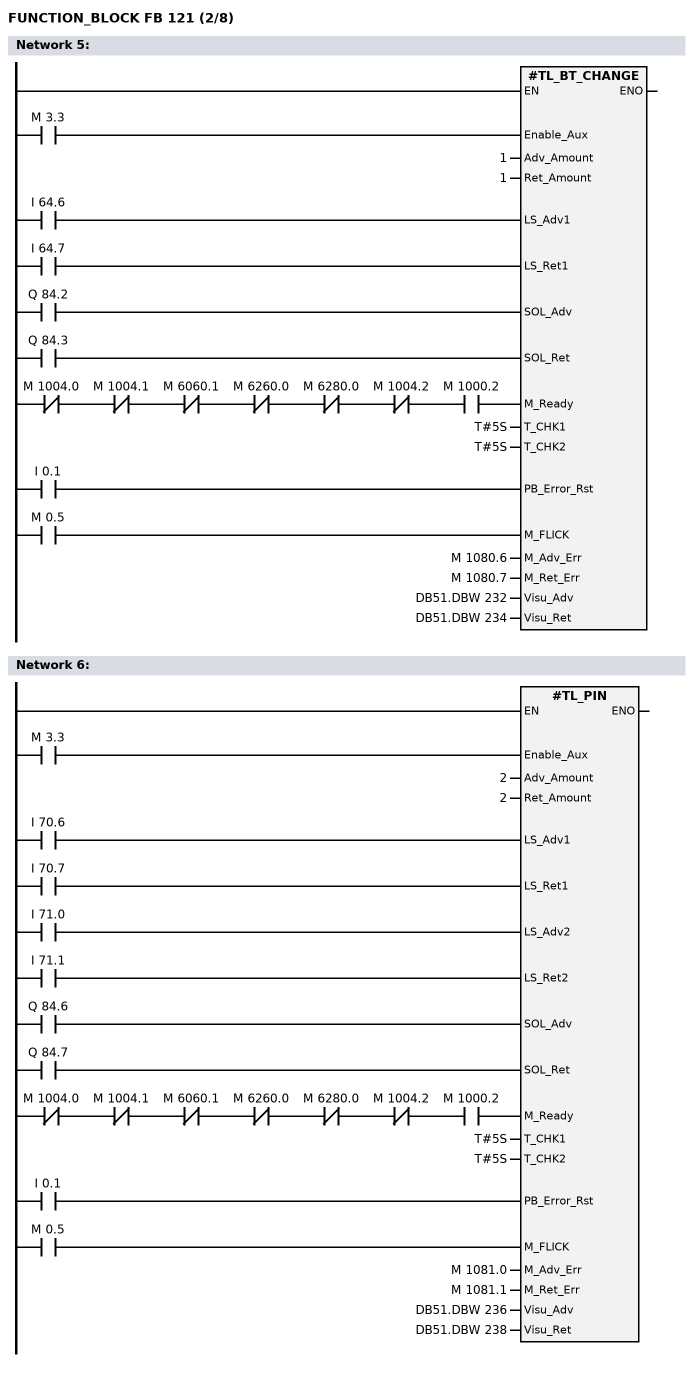

      A     M      3.3;
      =     L      0.0;
      BLD   103;
      A     I     64.6;
      =     L      0.1;
      BLD   103;
      A     I     64.7;
      =     L      0.2;
      BLD   103;
      A     Q     84.2;
      =     L      1.1;
      BLD   103;
      A     Q     84.3;
      =     L      1.2;
      BLD   103;
      AN    M   1004.0;
      AN    M   1004.1;
      AN    M   6060.1;
      AN    M   6260.0;
      AN    M   6280.0;
      AN    M   1004.2;
      A     M   1000.2;
      =     L      1.3;
      BLD   103;
      A     I      0.1;
      =     L      1.5;
      BLD   103;
      A     M      0.5;
      =     L      1.6;
      BLD   103;
      CALL #TL_BT_CHANGE (
           Enable_Aux               := L      0.0,
           Adv_Amount               := 1,
           Ret_Amount               := 1,
           LS_Adv1                  := L      0.1,
           LS_Ret1                  := L      0.2,
           SOL_Adv                  := L      1.1,
           SOL_Ret                  := L      1.2,
           M_Ready                  := L      1.3,
           T_CHK1                   := T#5S,
           T_CHK2                   := T#5S,
           PB_Error_Rst             := L      1.5,
           M_FLICK                  := L      1.6,
           M_Adv_Err                := M   1080.6,
           M_Ret_Err                := M   1080.7,
           Visu_Adv                 := DB51.DBW  232,
           Visu_Ret                 := DB51.DBW  234);
      NOP   0;
NETWORK
TITLE =

      A     M      3.3;
      =     L      0.0;
      BLD   103;
      A     I     70.6;
      =     L      0.1;
      BLD   103;
      A     I     70.7;
      =     L      0.2;
      BLD   103;
      A     I     71.0;
      =     L      0.3;
      BLD   103;
      A     I     71.1;
      =     L      0.4;
      BLD   103;
      A     Q     84.6;
      =     L      1.1;
      BLD   103;
      A     Q     84.7;
      =     L      1.2;
      BLD   103;
      AN    M   1004.0;
      AN    M   1004.1;
      AN    M   6060.1;
      AN    M   6260.0;
      AN    M   6280.0;
      AN    M   1004.2;
      A     M   1000.2;
      =     L      1.3;
      BLD   103;
      A     I      0.1;
      =     L      1.5;
      BLD   103;
      A     M      0.5;
      =     L      1.6;
      BLD   103;
      CALL #TL_PIN (
           Enable_Aux               := L      0.0,
           Adv_Amount               := 2,
           Ret_Amount               := 2,
           LS_Adv1                  := L      0.1,
           LS_Ret1                  := L      0.2,
           LS_Adv2                  := L      0.3,
           LS_Ret2                  := L      0.4,
           SOL_Adv                  := L      1.1,
           SOL_Ret                  := L      1.2,
           M_Ready                  := L      1.3,
           T_CHK1                   := T#5S,
           T_CHK2                   := T#5S,
           PB_Error_Rst             := L      1.5,
           M_FLICK                  := L      1.6,
           M_Adv_Err                := M   1081.0,
           M_Ret_Err                := M   1081.1,
           Visu_Adv                 := DB51.DBW  236,
           Visu_Ret                 := DB51.DBW  238);
      NOP   0;
NETWORK
TITLE =
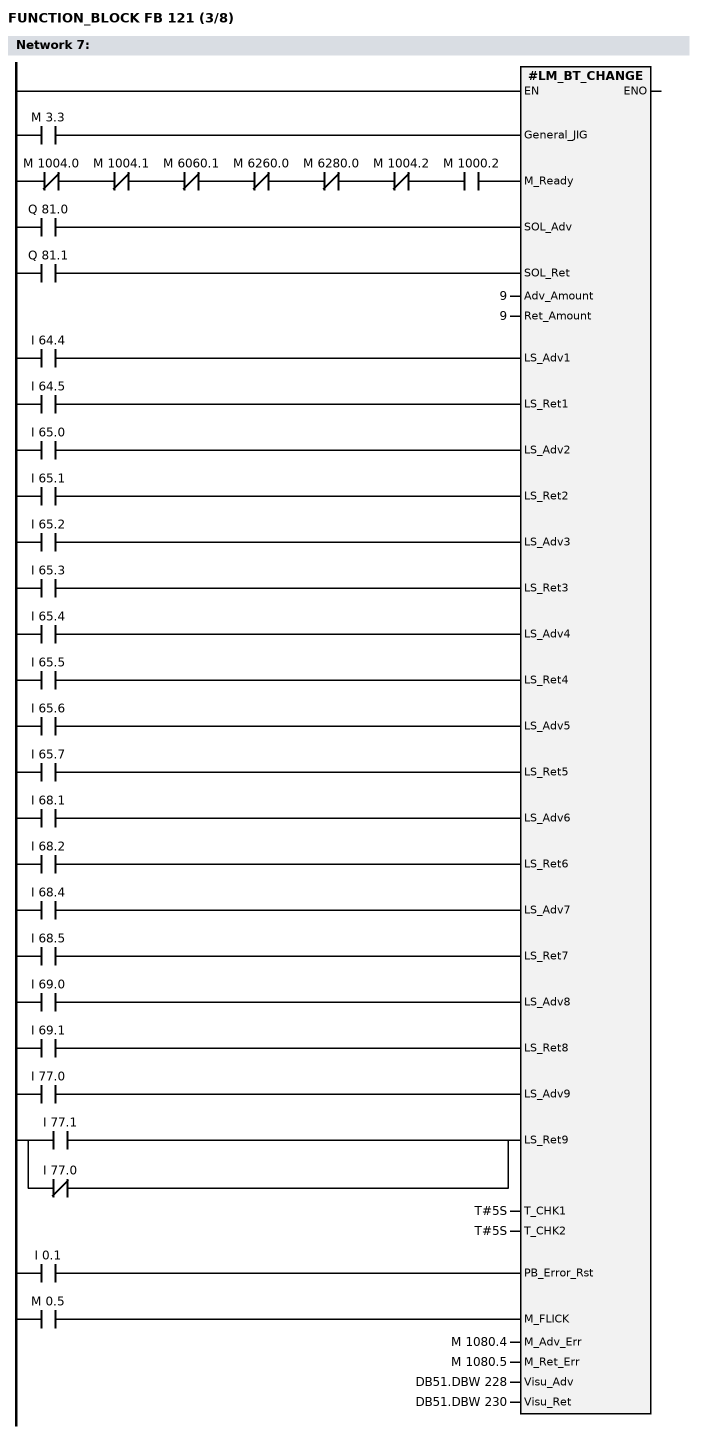

      A     M      3.3;
      =     L      0.0;
      BLD   103;
      AN    M   1004.0;
      AN    M   1004.1;
      AN    M   6060.1;
      AN    M   6260.0;
      AN    M   6280.0;
      AN    M   1004.2;
      A     M   1000.2;
      =     L      0.2;
      BLD   103;
      A     Q     81.0;
      =     L      0.3;
      BLD   103;
      A     Q     81.1;
      =     L      0.4;
      BLD   103;
      A     I     64.4;
      =     L      0.5;
      BLD   103;
      A     I     64.5;
      =     L      0.6;
      BLD   103;
      A     I     65.0;
      =     L      0.7;
      BLD   103;
      A     I     65.1;
      =     L      1.0;
      BLD   103;
      A     I     65.2;
      =     L      1.1;
      BLD   103;
      A     I     65.3;
      =     L      1.2;
      BLD   103;
      A     I     65.4;
      =     L      1.3;
      BLD   103;
      A     I     65.5;
      =     L      1.4;
      BLD   103;
      A     I     65.6;
      =     L      1.5;
      BLD   103;
      A     I     65.7;
      =     L      1.6;
      BLD   103;
      A     I     68.1;
      =     L      1.7;
      BLD   103;
      A     I     68.2;
      =     L      2.0;
      BLD   103;
      A     I     68.4;
      =     L      2.1;
      BLD   103;
      A     I     68.5;
      =     L      2.2;
      BLD   103;
      A     I     69.0;
      =     L      2.3;
      BLD   103;
      A     I     69.1;
      =     L      2.4;
      BLD   103;
      A     I     77.0;
      =     L      2.5;
      BLD   103;
      A(    ;
      O     I     77.1;
      ON    I     77.0;
      )     ;
      =     L      2.6;
      BLD   103;
      A     I      0.1;
      =     L      3.1;
      BLD   103;
      A     M      0.5;
      =     L      3.3;
      BLD   103;
      CALL #LM_BT_CHANGE (
           General_JIG              := L      0.0,
           M_Ready                  := L      0.2,
           SOL_Adv                  := L      0.3,
           SOL_Ret                  := L      0.4,
           Adv_Amount               := 9,
           Ret_Amount               := 9,
           LS_Adv1                  := L      0.5,
           LS_Ret1                  := L      0.6,
           LS_Adv2                  := L      0.7,
           LS_Ret2                  := L      1.0,
           LS_Adv3                  := L      1.1,
           LS_Ret3                  := L      1.2,
           LS_Adv4                  := L      1.3,
           LS_Ret4                  := L      1.4,
           LS_Adv5                  := L      1.5,
           LS_Ret5                  := L      1.6,
           LS_Adv6                  := L      1.7,
           LS_Ret6                  := L      2.0,
           LS_Adv7                  := L      2.1,
           LS_Ret7                  := L      2.2,
           LS_Adv8                  := L      2.3,
           LS_Ret8                  := L      2.4,
           LS_Adv9                  := L      2.5,
           LS_Ret9                  := L      2.6,
           T_CHK1                   := T#5S,
           T_CHK2                   := T#5S,
           PB_Error_Rst             := L      3.1,
           M_FLICK                  := L      3.3,
           M_Adv_Err                := M   1080.4,
           M_Ret_Err                := M   1080.5,
           Visu_Adv                 := DB51.DBW  228,
           Visu_Ret                 := DB51.DBW  230);
      NOP   0;
NETWORK
TITLE =
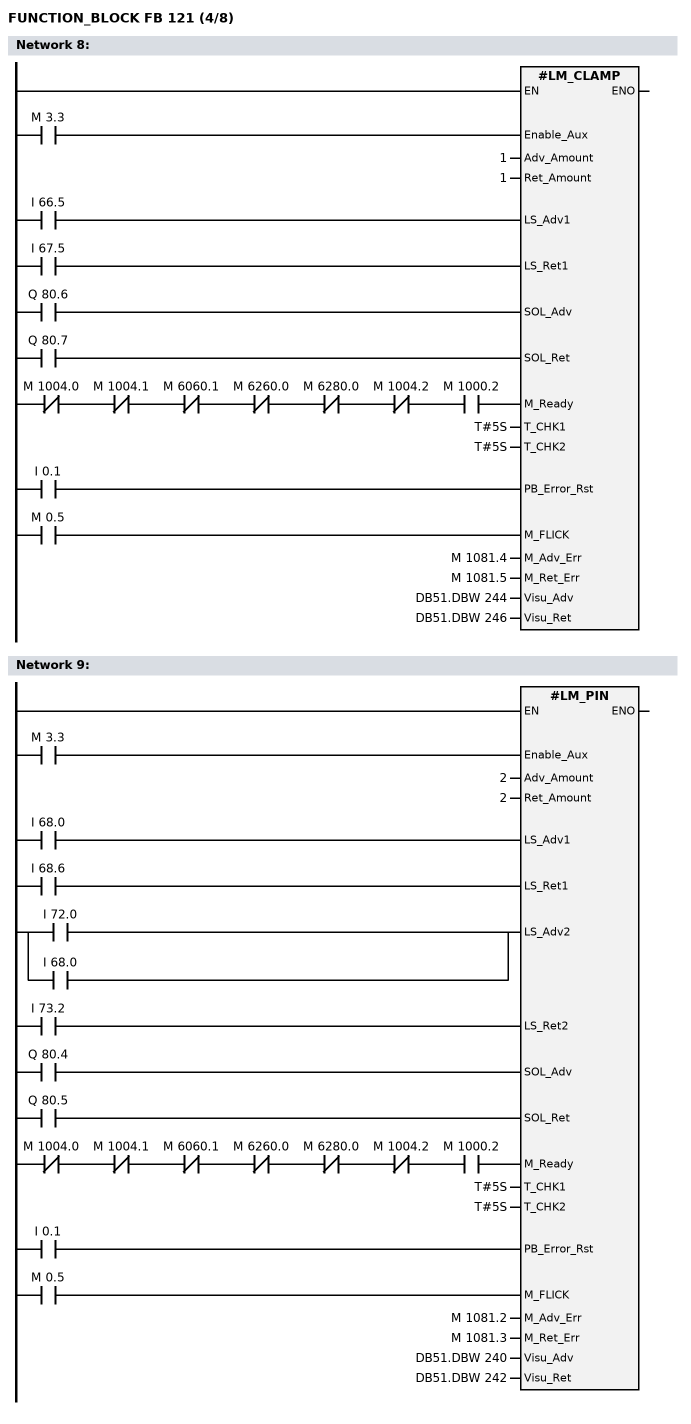

      A     M      3.3;
      =     L      0.0;
      BLD   103;
      A     I     66.5;
      =     L      0.1;
      BLD   103;
      A     I     67.5;
      =     L      0.2;
      BLD   103;
      A     Q     80.6;
      =     L      1.1;
      BLD   103;
      A     Q     80.7;
      =     L      1.2;
      BLD   103;
      AN    M   1004.0;
      AN    M   1004.1;
      AN    M   6060.1;
      AN    M   6260.0;
      AN    M   6280.0;
      AN    M   1004.2;
      A     M   1000.2;
      =     L      1.3;
      BLD   103;
      A     I      0.1;
      =     L      1.5;
      BLD   103;
      A     M      0.5;
      =     L      1.6;
      BLD   103;
      CALL #LM_CLAMP (
           Enable_Aux               := L      0.0,
           Adv_Amount               := 1,
           Ret_Amount               := 1,
           LS_Adv1                  := L      0.1,
           LS_Ret1                  := L      0.2,
           SOL_Adv                  := L      1.1,
           SOL_Ret                  := L      1.2,
           M_Ready                  := L      1.3,
           T_CHK1                   := T#5S,
           T_CHK2                   := T#5S,
           PB_Error_Rst             := L      1.5,
           M_FLICK                  := L      1.6,
           M_Adv_Err                := M   1081.4,
           M_Ret_Err                := M   1081.5,
           Visu_Adv                 := DB51.DBW  244,
           Visu_Ret                 := DB51.DBW  246);
      NOP   0;
NETWORK
TITLE =

      A     M      3.3;
      =     L      0.0;
      BLD   103;
      A     I     68.0;
      =     L      0.1;
      BLD   103;
      A     I     68.6;
      =     L      0.2;
      BLD   103;
      A(    ;
      O     I     72.0;
      O     I     68.0;
      )     ;
      =     L      0.3;
      BLD   103;
      A     I     73.2;
      =     L      0.4;
      BLD   103;
      A     Q     80.4;
      =     L      1.1;
      BLD   103;
      A     Q     80.5;
      =     L      1.2;
      BLD   103;
      AN    M   1004.0;
      AN    M   1004.1;
      AN    M   6060.1;
      AN    M   6260.0;
      AN    M   6280.0;
      AN    M   1004.2;
      A     M   1000.2;
      =     L      1.3;
      BLD   103;
      A     I      0.1;
      =     L      1.5;
      BLD   103;
      A     M      0.5;
      =     L      1.6;
      BLD   103;
      CALL #LM_PIN (
           Enable_Aux               := L      0.0,
           Adv_Amount               := 2,
           Ret_Amount               := 2,
           LS_Adv1                  := L      0.1,
           LS_Ret1                  := L      0.2,
           LS_Adv2                  := L      0.3,
           LS_Ret2                  := L      0.4,
           SOL_Adv                  := L      1.1,
           SOL_Ret                  := L      1.2,
           M_Ready                  := L      1.3,
           T_CHK1                   := T#5S,
           T_CHK2                   := T#5S,
           PB_Error_Rst             := L      1.5,
           M_FLICK                  := L      1.6,
           M_Adv_Err                := M   1081.2,
           M_Ret_Err                := M   1081.3,
           Visu_Adv                 := DB51.DBW  240,
           Visu_Ret                 := DB51.DBW  242);
      NOP   0;
NETWORK
TITLE =
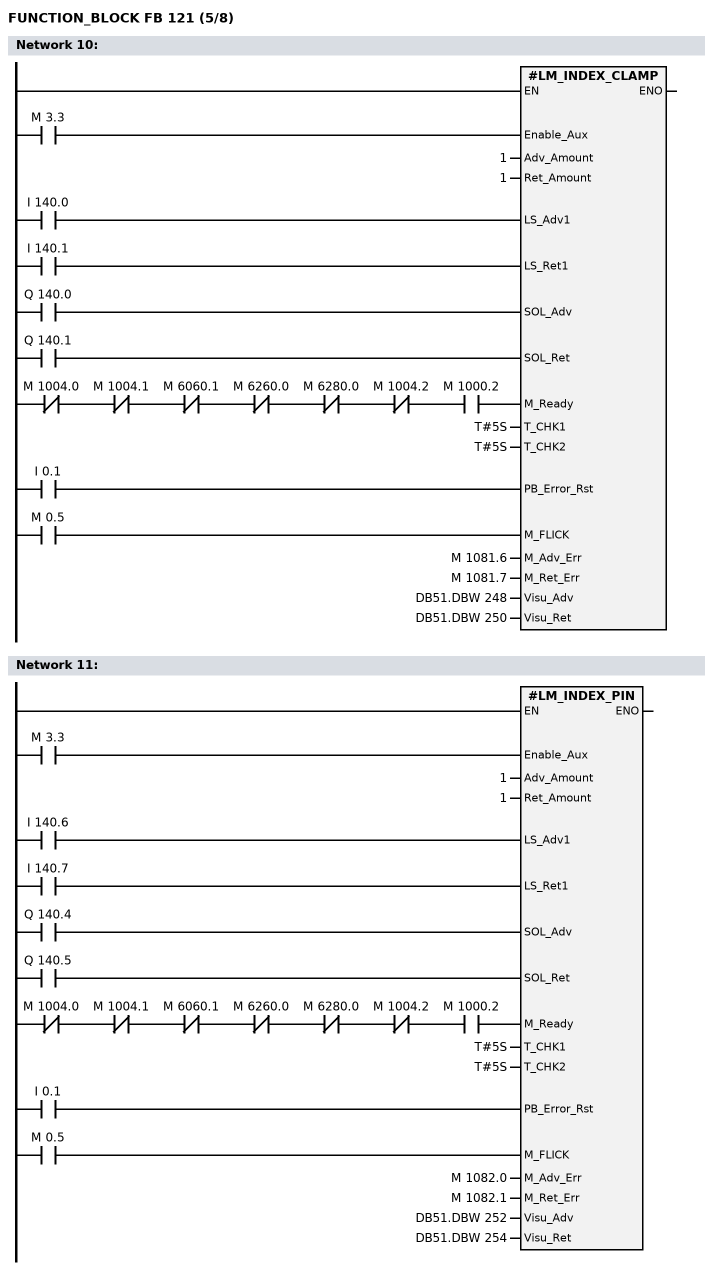

      A     M      3.3;
      =     L      0.0;
      BLD   103;
      A     I    140.0;
      =     L      0.1;
      BLD   103;
      A     I    140.1;
      =     L      0.2;
      BLD   103;
      A     Q    140.0;
      =     L      1.1;
      BLD   103;
      A     Q    140.1;
      =     L      1.2;
      BLD   103;
      AN    M   1004.0;
      AN    M   1004.1;
      AN    M   6060.1;
      AN    M   6260.0;
      AN    M   6280.0;
      AN    M   1004.2;
      A     M   1000.2;
      =     L      1.3;
      BLD   103;
      A     I      0.1;
      =     L      1.5;
      BLD   103;
      A     M      0.5;
      =     L      1.6;
      BLD   103;
      CALL #LM_INDEX_CLAMP (
           Enable_Aux               := L      0.0,
           Adv_Amount               := 1,
           Ret_Amount               := 1,
           LS_Adv1                  := L      0.1,
           LS_Ret1                  := L      0.2,
           SOL_Adv                  := L      1.1,
           SOL_Ret                  := L      1.2,
           M_Ready                  := L      1.3,
           T_CHK1                   := T#5S,
           T_CHK2                   := T#5S,
           PB_Error_Rst             := L      1.5,
           M_FLICK                  := L      1.6,
           M_Adv_Err                := M   1081.6,
           M_Ret_Err                := M   1081.7,
           Visu_Adv                 := DB51.DBW  248,
           Visu_Ret                 := DB51.DBW  250);
      NOP   0;
NETWORK
TITLE =

      A     M      3.3;
      =     L      0.0;
      BLD   103;
      A     I    140.6;
      =     L      0.1;
      BLD   103;
      A     I    140.7;
      =     L      0.2;
      BLD   103;
      A     Q    140.4;
      =     L      1.1;
      BLD   103;
      A     Q    140.5;
      =     L      1.2;
      BLD   103;
      AN    M   1004.0;
      AN    M   1004.1;
      AN    M   6060.1;
      AN    M   6260.0;
      AN    M   6280.0;
      AN    M   1004.2;
      A     M   1000.2;
      =     L      1.3;
      BLD   103;
      A     I      0.1;
      =     L      1.5;
      BLD   103;
      A     M      0.5;
      =     L      1.6;
      BLD   103;
      CALL #LM_INDEX_PIN (
           Enable_Aux               := L      0.0,
           Adv_Amount               := 1,
           Ret_Amount               := 1,
           LS_Adv1                  := L      0.1,
           LS_Ret1                  := L      0.2,
           SOL_Adv                  := L      1.1,
           SOL_Ret                  := L      1.2,
           M_Ready                  := L      1.3,
           T_CHK1                   := T#5S,
           T_CHK2                   := T#5S,
           PB_Error_Rst             := L      1.5,
           M_FLICK                  := L      1.6,
           M_Adv_Err                := M   1082.0,
           M_Ret_Err                := M   1082.1,
           Visu_Adv                 := DB51.DBW  252,
           Visu_Ret                 := DB51.DBW  254);
      NOP   0;
NETWORK
TITLE =#711 INR PLT LS이상

NETWORK
TITLE =
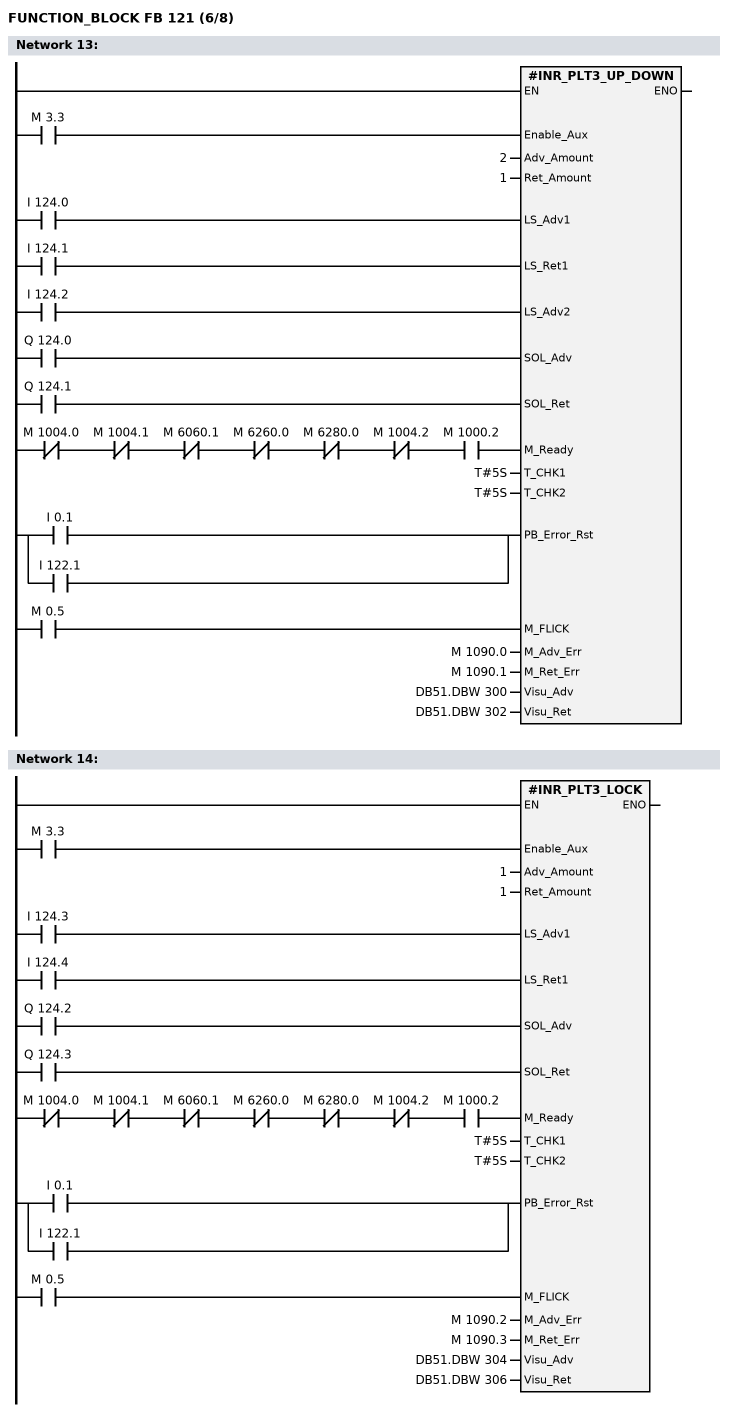

      A     M      3.3;
      =     L      0.0;
      BLD   103;
      A     I    124.0;
      =     L      0.1;
      BLD   103;
      A     I    124.1;
      =     L      0.2;
      BLD   103;
      A     I    124.2;
      =     L      0.3;
      BLD   103;
      A     Q    124.0;
      =     L      1.1;
      BLD   103;
      A     Q    124.1;
      =     L      1.2;
      BLD   103;
      AN    M   1004.0;
      AN    M   1004.1;
      AN    M   6060.1;
      AN    M   6260.0;
      AN    M   6280.0;
      AN    M   1004.2;
      A     M   1000.2;
      =     L      1.3;
      BLD   103;
      A(    ;
      O     I      0.1;
      O     I    122.1;
      )     ;
      =     L      1.5;
      BLD   103;
      A     M      0.5;
      =     L      1.6;
      BLD   103;
      CALL #INR_PLT3_UP_DOWN (
           Enable_Aux               := L      0.0,
           Adv_Amount               := 2,
           Ret_Amount               := 1,
           LS_Adv1                  := L      0.1,
           LS_Ret1                  := L      0.2,
           LS_Adv2                  := L      0.3,
           SOL_Adv                  := L      1.1,
           SOL_Ret                  := L      1.2,
           M_Ready                  := L      1.3,
           T_CHK1                   := T#5S,
           T_CHK2                   := T#5S,
           PB_Error_Rst             := L      1.5,
           M_FLICK                  := L      1.6,
           M_Adv_Err                := M   1090.0,
           M_Ret_Err                := M   1090.1,
           Visu_Adv                 := DB51.DBW  300,
           Visu_Ret                 := DB51.DBW  302);
      NOP   0;
NETWORK
TITLE =

      A     M      3.3;
      =     L      0.0;
      BLD   103;
      A     I    124.3;
      =     L      0.1;
      BLD   103;
      A     I    124.4;
      =     L      0.2;
      BLD   103;
      A     Q    124.2;
      =     L      1.1;
      BLD   103;
      A     Q    124.3;
      =     L      1.2;
      BLD   103;
      AN    M   1004.0;
      AN    M   1004.1;
      AN    M   6060.1;
      AN    M   6260.0;
      AN    M   6280.0;
      AN    M   1004.2;
      A     M   1000.2;
      =     L      1.3;
      BLD   103;
      A(    ;
      O     I      0.1;
      O     I    122.1;
      )     ;
      =     L      1.5;
      BLD   103;
      A     M      0.5;
      =     L      1.6;
      BLD   103;
      CALL #INR_PLT3_LOCK (
           Enable_Aux               := L      0.0,
           Adv_Amount               := 1,
           Ret_Amount               := 1,
           LS_Adv1                  := L      0.1,
           LS_Ret1                  := L      0.2,
           SOL_Adv                  := L      1.1,
           SOL_Ret                  := L      1.2,
           M_Ready                  := L      1.3,
           T_CHK1                   := T#5S,
           T_CHK2                   := T#5S,
           PB_Error_Rst             := L      1.5,
           M_FLICK                  := L      1.6,
           M_Adv_Err                := M   1090.2,
           M_Ret_Err                := M   1090.3,
           Visu_Adv                 := DB51.DBW  304,
           Visu_Ret                 := DB51.DBW  306);
      NOP   0;
NETWORK
TITLE =
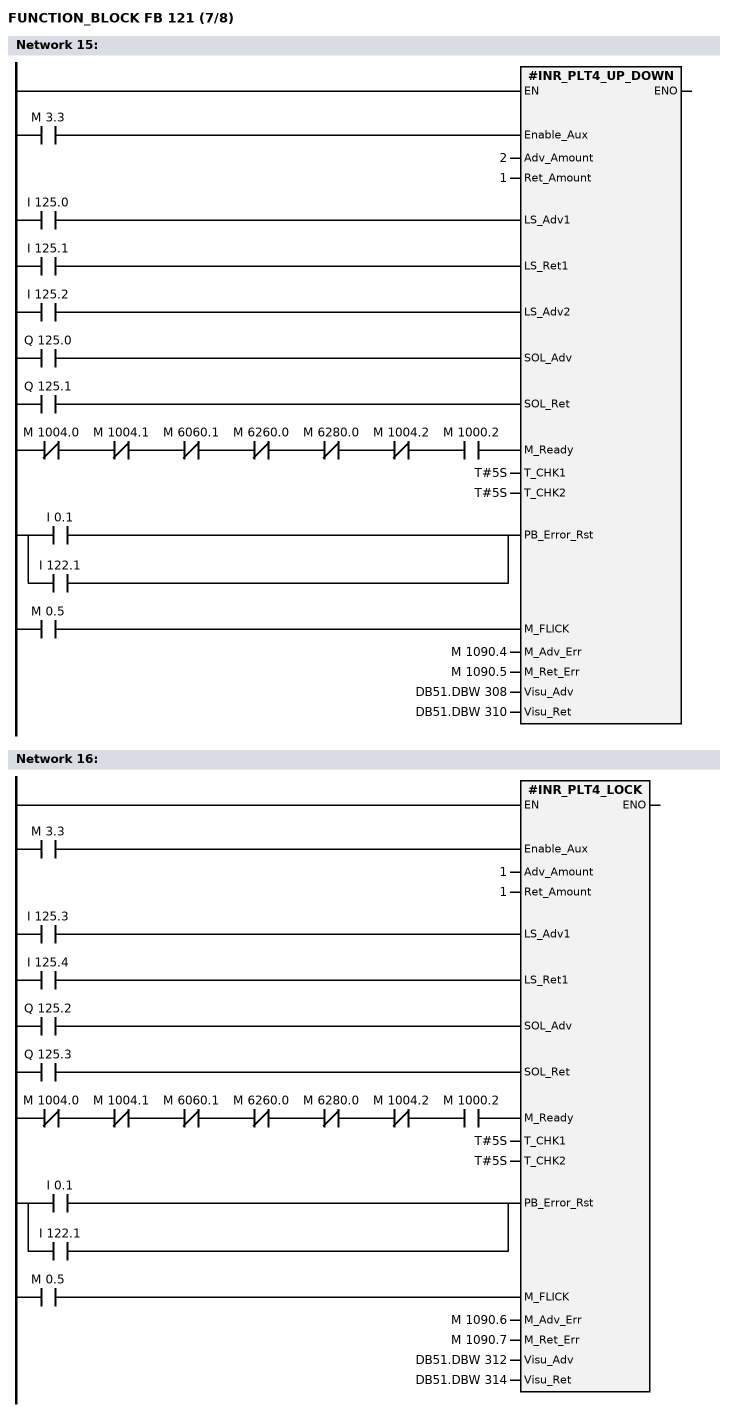

      A     M      3.3;
      =     L      0.0;
      BLD   103;
      A     I    125.0;
      =     L      0.1;
      BLD   103;
      A     I    125.1;
      =     L      0.2;
      BLD   103;
      A     I    125.2;
      =     L      0.3;
      BLD   103;
      A     Q    125.0;
      =     L      1.1;
      BLD   103;
      A     Q    125.1;
      =     L      1.2;
      BLD   103;
      AN    M   1004.0;
      AN    M   1004.1;
      AN    M   6060.1;
      AN    M   6260.0;
      AN    M   6280.0;
      AN    M   1004.2;
      A     M   1000.2;
      =     L      1.3;
      BLD   103;
      A(    ;
      O     I      0.1;
      O     I    122.1;
      )     ;
      =     L      1.5;
      BLD   103;
      A     M      0.5;
      =     L      1.6;
      BLD   103;
      CALL #INR_PLT4_UP_DOWN (
           Enable_Aux               := L      0.0,
           Adv_Amount               := 2,
           Ret_Amount               := 1,
           LS_Adv1                  := L      0.1,
           LS_Ret1                  := L      0.2,
           LS_Adv2                  := L      0.3,
           SOL_Adv                  := L      1.1,
           SOL_Ret                  := L      1.2,
           M_Ready                  := L      1.3,
           T_CHK1                   := T#5S,
           T_CHK2                   := T#5S,
           PB_Error_Rst             := L      1.5,
           M_FLICK                  := L      1.6,
           M_Adv_Err                := M   1090.4,
           M_Ret_Err                := M   1090.5,
           Visu_Adv                 := DB51.DBW  308,
           Visu_Ret                 := DB51.DBW  310);
      NOP   0;
NETWORK
TITLE =

      A     M      3.3;
      =     L      0.0;
      BLD   103;
      A     I    125.3;
      =     L      0.1;
      BLD   103;
      A     I    125.4;
      =     L      0.2;
      BLD   103;
      A     Q    125.2;
      =     L      1.1;
      BLD   103;
      A     Q    125.3;
      =     L      1.2;
      BLD   103;
      AN    M   1004.0;
      AN    M   1004.1;
      AN    M   6060.1;
      AN    M   6260.0;
      AN    M   6280.0;
      AN    M   1004.2;
      A     M   1000.2;
      =     L      1.3;
      BLD   103;
      A(    ;
      O     I      0.1;
      O     I    122.1;
      )     ;
      =     L      1.5;
      BLD   103;
      A     M      0.5;
      =     L      1.6;
      BLD   103;
      CALL #INR_PLT4_LOCK (
           Enable_Aux               := L      0.0,
           Adv_Amount               := 1,
           Ret_Amount               := 1,
           LS_Adv1                  := L      0.1,
           LS_Ret1                  := L      0.2,
           SOL_Adv                  := L      1.1,
           SOL_Ret                  := L      1.2,
           M_Ready                  := L      1.3,
           T_CHK1                   := T#5S,
           T_CHK2                   := T#5S,
           PB_Error_Rst             := L      1.5,
           M_FLICK                  := L      1.6,
           M_Adv_Err                := M   1090.6,
           M_Ret_Err                := M   1090.7,
           Visu_Adv                 := DB51.DBW  312,
           Visu_Ret                 := DB51.DBW  314);
      NOP   0;
NETWORK
TITLE =
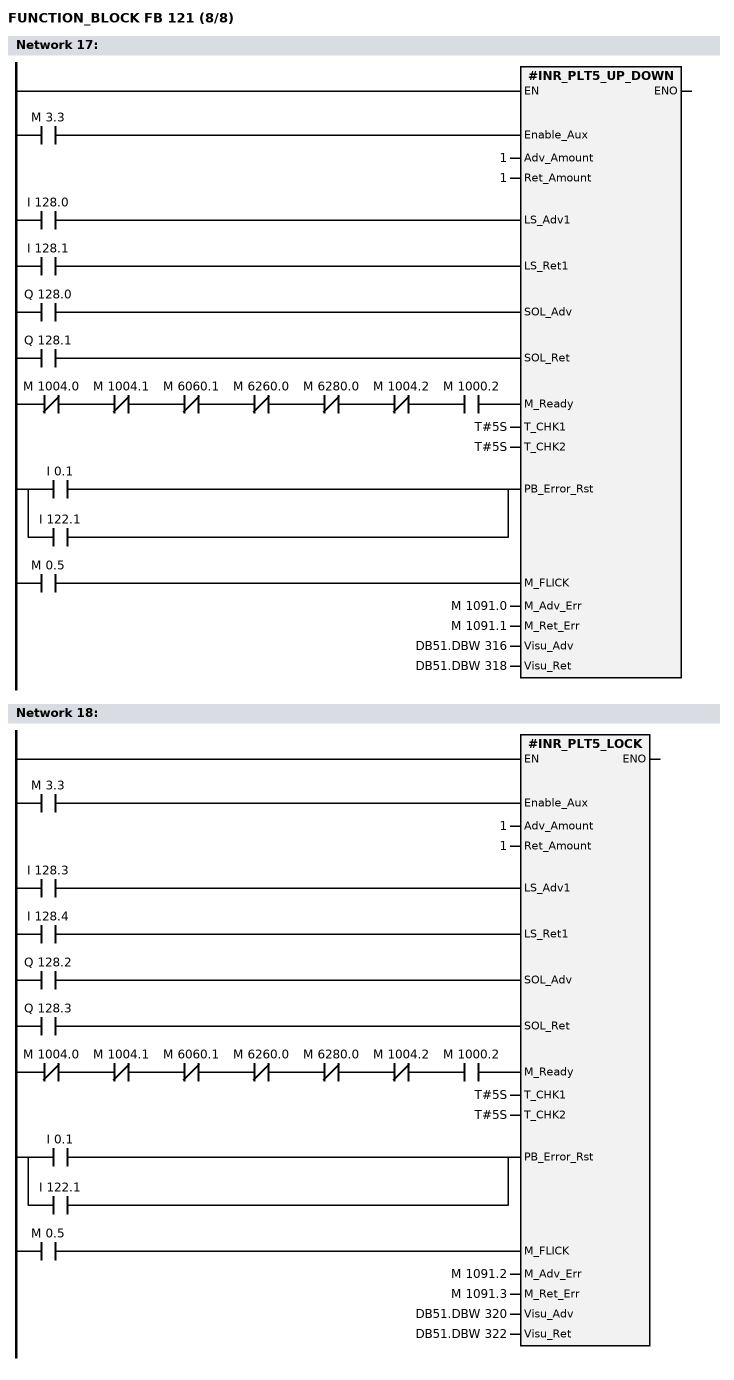

      A     M      3.3;
      =     L      0.0;
      BLD   103;
      A     I    128.0;
      =     L      0.1;
      BLD   103;
      A     I    128.1;
      =     L      0.2;
      BLD   103;
      A     Q    128.0;
      =     L      1.1;
      BLD   103;
      A     Q    128.1;
      =     L      1.2;
      BLD   103;
      AN    M   1004.0;
      AN    M   1004.1;
      AN    M   6060.1;
      AN    M   6260.0;
      AN    M   6280.0;
      AN    M   1004.2;
      A     M   1000.2;
      =     L      1.3;
      BLD   103;
      A(    ;
      O     I      0.1;
      O     I    122.1;
      )     ;
      =     L      1.5;
      BLD   103;
      A     M      0.5;
      =     L      1.6;
      BLD   103;
      CALL #INR_PLT5_UP_DOWN (
           Enable_Aux               := L      0.0,
           Adv_Amount               := 1,
           Ret_Amount               := 1,
           LS_Adv1                  := L      0.1,
           LS_Ret1                  := L      0.2,
           SOL_Adv                  := L      1.1,
           SOL_Ret                  := L      1.2,
           M_Ready                  := L      1.3,
           T_CHK1                   := T#5S,
           T_CHK2                   := T#5S,
           PB_Error_Rst             := L      1.5,
           M_FLICK                  := L      1.6,
           M_Adv_Err                := M   1091.0,
           M_Ret_Err                := M   1091.1,
           Visu_Adv                 := DB51.DBW  316,
           Visu_Ret                 := DB51.DBW  318);
      NOP   0;
NETWORK
TITLE =

      A     M      3.3;
      =     L      0.0;
      BLD   103;
      A     I    128.3;
      =     L      0.1;
      BLD   103;
      A     I    128.4;
      =     L      0.2;
      BLD   103;
      A     Q    128.2;
      =     L      1.1;
      BLD   103;
      A     Q    128.3;
      =     L      1.2;
      BLD   103;
      AN    M   1004.0;
      AN    M   1004.1;
      AN    M   6060.1;
      AN    M   6260.0;
      AN    M   6280.0;
      AN    M   1004.2;
      A     M   1000.2;
      =     L      1.3;
      BLD   103;
      A(    ;
      O     I      0.1;
      O     I    122.1;
      )     ;
      =     L      1.5;
      BLD   103;
      A     M      0.5;
      =     L      1.6;
      BLD   103;
      CALL #INR_PLT5_LOCK (
           Enable_Aux               := L      0.0,
           Adv_Amount               := 1,
           Ret_Amount               := 1,
           LS_Adv1                  := L      0.1,
           LS_Ret1                  := L      0.2,
           SOL_Adv                  := L      1.1,
           SOL_Ret                  := L      1.2,
           M_Ready                  := L      1.3,
           T_CHK1                   := T#5S,
           T_CHK2                   := T#5S,
           PB_Error_Rst             := L      1.5,
           M_FLICK                  := L      1.6,
           M_Adv_Err                := M   1091.2,
           M_Ret_Err                := M   1091.3,
           Visu_Adv                 := DB51.DBW  320,
           Visu_Ret                 := DB51.DBW  322);
      NOP   0;
END_FUNCTION_BLOCK

DATA_BLOCK DB 121
TITLE =
VERSION : 0.0

 FB 121
BEGIN
   INDEX_LOCK.Enable_Aux := FALSE;
   INDEX_LOCK.Adv_Amount := 0;
   INDEX_LOCK.Ret_Amount := 0;
   INDEX_LOCK.LS_Adv1 := FALSE;
   INDEX_LOCK.LS_Ret1 := FALSE;
   INDEX_LOCK.LS_Adv2 := FALSE;
   INDEX_LOCK.LS_Ret2 := FALSE;
   INDEX_LOCK.LS_Adv3 := FALSE;
   INDEX_LOCK.LS_Ret3 := FALSE;
   INDEX_LOCK.LS_Adv4 := FALSE;
   INDEX_LOCK.LS_Ret4 := FALSE;
   INDEX_LOCK.SOL_Adv := FALSE;
   INDEX_LOCK.SOL_Ret := FALSE;
   INDEX_LOCK.M_Ready := FALSE;
   INDEX_LOCK.T_CHK1 := T#0MS;
   INDEX_LOCK.T_CHK2 := T#0MS;
   INDEX_LOCK.PB_Lamp_CHK := FALSE;
   INDEX_LOCK.PB_Error_Rst := FALSE;
   INDEX_LOCK.M_FLICK := FALSE;
   INDEX_LOCK.M_Adv_Err := FALSE;
   INDEX_LOCK.M_Ret_Err := FALSE;
   INDEX_LOCK.LP_Adv := FALSE;
   INDEX_LOCK.LP_Ret := FALSE;
   INDEX_LOCK.Visu_Adv := W#16#0;
   INDEX_LOCK.Visu_Ret := W#16#0;
   INDEX_LOCK.Error_T1.IN := FALSE;
   INDEX_LOCK.Error_T1.PT := T#0MS;
   INDEX_LOCK.Error_T1.Q := FALSE;
   INDEX_LOCK.Error_T1.ET := T#0MS;
   INDEX_LOCK.Error_T1.STATE := B#16#0;
   INDEX_LOCK.Error_T1.STIME := T#0MS;
   INDEX_LOCK.Error_T1.ATIME := T#0MS;
   INDEX_LOCK.Error_T2.IN := FALSE;
   INDEX_LOCK.Error_T2.PT := T#0MS;
   INDEX_LOCK.Error_T2.Q := FALSE;
   INDEX_LOCK.Error_T2.ET := T#0MS;
   INDEX_LOCK.Error_T2.STATE := B#16#0;
   INDEX_LOCK.Error_T2.STIME := T#0MS;
   INDEX_LOCK.Error_T2.ATIME := T#0MS;
   INDEX_LOCK.CHK_Aux1 := FALSE;
   INDEX_LOCK.CHK_Aux2 := FALSE;
   INDEX_LOCK.Error_T1_DN := FALSE;
   INDEX_LOCK.Error_T2_DN := FALSE;
   INDEX_LOCK.Adv_Memo := FALSE;
   INDEX_LOCK.Visu_Adv_Arr[0] := FALSE;
   INDEX_LOCK.Visu_Adv_Arr[1] := FALSE;
   INDEX_LOCK.Visu_Adv_Arr[2] := FALSE;
   INDEX_LOCK.Visu_Adv_Arr[3] := FALSE;
   INDEX_LOCK.Visu_Adv_Arr[4] := FALSE;
   INDEX_LOCK.Visu_Adv_Arr[5] := FALSE;
   INDEX_LOCK.Visu_Adv_Arr[6] := FALSE;
   INDEX_LOCK.Visu_Adv_Arr[7] := FALSE;
   INDEX_LOCK.Visu_Adv_Arr[8] := FALSE;
   INDEX_LOCK.Visu_Adv_Arr[9] := FALSE;
   INDEX_LOCK.Visu_Adv_Arr[10] := FALSE;
   INDEX_LOCK.Visu_Adv_Arr[11] := FALSE;
   INDEX_LOCK.Visu_Adv_Arr[12] := FALSE;
   INDEX_LOCK.Visu_Adv_Arr[13] := FALSE;
   INDEX_LOCK.Visu_Adv_Arr[14] := FALSE;
   INDEX_LOCK.Visu_Adv_Arr[15] := FALSE;
   INDEX_LOCK.Visu_Ret_Arr[0] := FALSE;
   INDEX_LOCK.Visu_Ret_Arr[1] := FALSE;
   INDEX_LOCK.Visu_Ret_Arr[2] := FALSE;
   INDEX_LOCK.Visu_Ret_Arr[3] := FALSE;
   INDEX_LOCK.Visu_Ret_Arr[4] := FALSE;
   INDEX_LOCK.Visu_Ret_Arr[5] := FALSE;
   INDEX_LOCK.Visu_Ret_Arr[6] := FALSE;
   INDEX_LOCK.Visu_Ret_Arr[7] := FALSE;
   INDEX_LOCK.Visu_Ret_Arr[8] := FALSE;
   INDEX_LOCK.Visu_Ret_Arr[9] := FALSE;
   INDEX_LOCK.Visu_Ret_Arr[10] := FALSE;
   INDEX_LOCK.Visu_Ret_Arr[11] := FALSE;
   INDEX_LOCK.Visu_Ret_Arr[12] := FALSE;
   INDEX_LOCK.Visu_Ret_Arr[13] := FALSE;
   INDEX_LOCK.Visu_Ret_Arr[14] := FALSE;
   INDEX_LOCK.Visu_Ret_Arr[15] := FALSE;
   INDEX_LOCK.BLK_Move_Ret := 0;
   INDEX_LOCK.Enable := FALSE;
   INDEX_LOCK.Adv_End := FALSE;
   INDEX_LOCK.Ret_End := FALSE;
   TL_BT_CHANGE.Enable_Aux := FALSE;
   TL_BT_CHANGE.Adv_Amount := 0;
   TL_BT_CHANGE.Ret_Amount := 0;
   TL_BT_CHANGE.LS_Adv1 := FALSE;
   TL_BT_CHANGE.LS_Ret1 := FALSE;
   TL_BT_CHANGE.LS_Adv2 := FALSE;
   TL_BT_CHANGE.LS_Ret2 := FALSE;
   TL_BT_CHANGE.LS_Adv3 := FALSE;
   TL_BT_CHANGE.LS_Ret3 := FALSE;
   TL_BT_CHANGE.LS_Adv4 := FALSE;
   TL_BT_CHANGE.LS_Ret4 := FALSE;
   TL_BT_CHANGE.SOL_Adv := FALSE;
   TL_BT_CHANGE.SOL_Ret := FALSE;
   TL_BT_CHANGE.M_Ready := FALSE;
   TL_BT_CHANGE.T_CHK1 := T#0MS;
   TL_BT_CHANGE.T_CHK2 := T#0MS;
   TL_BT_CHANGE.PB_Lamp_CHK := FALSE;
   TL_BT_CHANGE.PB_Error_Rst := FALSE;
   TL_BT_CHANGE.M_FLICK := FALSE;
   TL_BT_CHANGE.M_Adv_Err := FALSE;
   TL_BT_CHANGE.M_Ret_Err := FALSE;
   TL_BT_CHANGE.LP_Adv := FALSE;
   TL_BT_CHANGE.LP_Ret := FALSE;
   TL_BT_CHANGE.Visu_Adv := W#16#0;
   TL_BT_CHANGE.Visu_Ret := W#16#0;
   TL_BT_CHANGE.Error_T1.IN := FALSE;
   TL_BT_CHANGE.Error_T1.PT := T#0MS;
   TL_BT_CHANGE.Error_T1.Q := FALSE;
   TL_BT_CHANGE.Error_T1.ET := T#0MS;
   TL_BT_CHANGE.Error_T1.STATE := B#16#0;
   TL_BT_CHANGE.Error_T1.STIME := T#0MS;
   TL_BT_CHANGE.Error_T1.ATIME := T#0MS;
   TL_BT_CHANGE.Error_T2.IN := FALSE;
   TL_BT_CHANGE.Error_T2.PT := T#0MS;
   TL_BT_CHANGE.Error_T2.Q := FALSE;
   TL_BT_CHANGE.Error_T2.ET := T#0MS;
   TL_BT_CHANGE.Error_T2.STATE := B#16#0;
   TL_BT_CHANGE.Error_T2.STIME := T#0MS;
   TL_BT_CHANGE.Error_T2.ATIME := T#0MS;
   TL_BT_CHANGE.CHK_Aux1 := FALSE;
   TL_BT_CHANGE.CHK_Aux2 := FALSE;
   TL_BT_CHANGE.Error_T1_DN := FALSE;
   TL_BT_CHANGE.Error_T2_DN := FALSE;
   TL_BT_CHANGE.Adv_Memo := FALSE;
   TL_BT_CHANGE.Visu_Adv_Arr[0] := FALSE;
   TL_BT_CHANGE.Visu_Adv_Arr[1] := FALSE;
   TL_BT_CHANGE.Visu_Adv_Arr[2] := FALSE;
   TL_BT_CHANGE.Visu_Adv_Arr[3] := FALSE;
   TL_BT_CHANGE.Visu_Adv_Arr[4] := FALSE;
   TL_BT_CHANGE.Visu_Adv_Arr[5] := FALSE;
   TL_BT_CHANGE.Visu_Adv_Arr[6] := FALSE;
   TL_BT_CHANGE.Visu_Adv_Arr[7] := FALSE;
   TL_BT_CHANGE.Visu_Adv_Arr[8] := FALSE;
   TL_BT_CHANGE.Visu_Adv_Arr[9] := FALSE;
   TL_BT_CHANGE.Visu_Adv_Arr[10] := FALSE;
   TL_BT_CHANGE.Visu_Adv_Arr[11] := FALSE;
   TL_BT_CHANGE.Visu_Adv_Arr[12] := FALSE;
   TL_BT_CHANGE.Visu_Adv_Arr[13] := FALSE;
   TL_BT_CHANGE.Visu_Adv_Arr[14] := FALSE;
   TL_BT_CHANGE.Visu_Adv_Arr[15] := FALSE;
   TL_BT_CHANGE.Visu_Ret_Arr[0] := FALSE;
   TL_BT_CHANGE.Visu_Ret_Arr[1] := FALSE;
   TL_BT_CHANGE.Visu_Ret_Arr[2] := FALSE;
   TL_BT_CHANGE.Visu_Ret_Arr[3] := FALSE;
   TL_BT_CHANGE.Visu_Ret_Arr[4] := FALSE;
   TL_BT_CHANGE.Visu_Ret_Arr[5] := FALSE;
   TL_BT_CHANGE.Visu_Ret_Arr[6] := FALSE;
   TL_BT_CHANGE.Visu_Ret_Arr[7] := FALSE;
   TL_BT_CHANGE.Visu_Ret_Arr[8] := FALSE;
   TL_BT_CHANGE.Visu_Ret_Arr[9] := FALSE;
   TL_BT_CHANGE.Visu_Ret_Arr[10] := FALSE;
   TL_BT_CHANGE.Visu_Ret_Arr[11] := FALSE;
   TL_BT_CHANGE.Visu_Ret_Arr[12] := FALSE;
   TL_BT_CHANGE.Visu_Ret_Arr[13] := FALSE;
   TL_BT_CHANGE.Visu_Ret_Arr[14] := FALSE;
   TL_BT_CHANGE.Visu_Ret_Arr[15] := FALSE;
   TL_BT_CHANGE.BLK_Move_Ret := 0;
   TL_BT_CHANGE.Enable := FALSE;
   TL_BT_CHANGE.Adv_End := FALSE;
   TL_BT_CHANGE.Ret_End := FALSE;
   TL_PIN.Enable_Aux := FALSE;
   TL_PIN.Adv_Amount := 0;
   TL_PIN.Ret_Amount := 0;
   TL_PIN.LS_Adv1 := FALSE;
   TL_PIN.LS_Ret1 := FALSE;
   TL_PIN.LS_Adv2 := FALSE;
   TL_PIN.LS_Ret2 := FALSE;
   TL_PIN.LS_Adv3 := FALSE;
   TL_PIN.LS_Ret3 := FALSE;
   TL_PIN.LS_Adv4 := FALSE;
   TL_PIN.LS_Ret4 := FALSE;
   TL_PIN.SOL_Adv := FALSE;
   TL_PIN.SOL_Ret := FALSE;
   TL_PIN.M_Ready := FALSE;
   TL_PIN.T_CHK1 := T#0MS;
   TL_PIN.T_CHK2 := T#0MS;
   TL_PIN.PB_Lamp_CHK := FALSE;
   TL_PIN.PB_Error_Rst := FALSE;
   TL_PIN.M_FLICK := FALSE;
   TL_PIN.M_Adv_Err := FALSE;
   TL_PIN.M_Ret_Err := FALSE;
   TL_PIN.LP_Adv := FALSE;
   TL_PIN.LP_Ret := FALSE;
   TL_PIN.Visu_Adv := W#16#0;
   TL_PIN.Visu_Ret := W#16#0;
   TL_PIN.Error_T1.IN := FALSE;
   TL_PIN.Error_T1.PT := T#0MS;
   TL_PIN.Error_T1.Q := FALSE;
   TL_PIN.Error_T1.ET := T#0MS;
   TL_PIN.Error_T1.STATE := B#16#0;
   TL_PIN.Error_T1.STIME := T#0MS;
   TL_PIN.Error_T1.ATIME := T#0MS;
   TL_PIN.Error_T2.IN := FALSE;
   TL_PIN.Error_T2.PT := T#0MS;
   TL_PIN.Error_T2.Q := FALSE;
   TL_PIN.Error_T2.ET := T#0MS;
   TL_PIN.Error_T2.STATE := B#16#0;
   TL_PIN.Error_T2.STIME := T#0MS;
   TL_PIN.Error_T2.ATIME := T#0MS;
   TL_PIN.CHK_Aux1 := FALSE;
   TL_PIN.CHK_Aux2 := FALSE;
   TL_PIN.Error_T1_DN := FALSE;
   TL_PIN.Error_T2_DN := FALSE;
   TL_PIN.Adv_Memo := FALSE;
   TL_PIN.Visu_Adv_Arr[0] := FALSE;
   TL_PIN.Visu_Adv_Arr[1] := FALSE;
   TL_PIN.Visu_Adv_Arr[2] := FALSE;
   TL_PIN.Visu_Adv_Arr[3] := FALSE;
   TL_PIN.Visu_Adv_Arr[4] := FALSE;
   TL_PIN.Visu_Adv_Arr[5] := FALSE;
   TL_PIN.Visu_Adv_Arr[6] := FALSE;
   TL_PIN.Visu_Adv_Arr[7] := FALSE;
   TL_PIN.Visu_Adv_Arr[8] := FALSE;
   TL_PIN.Visu_Adv_Arr[9] := FALSE;
   TL_PIN.Visu_Adv_Arr[10] := FALSE;
   TL_PIN.Visu_Adv_Arr[11] := FALSE;
   TL_PIN.Visu_Adv_Arr[12] := FALSE;
   TL_PIN.Visu_Adv_Arr[13] := FALSE;
   TL_PIN.Visu_Adv_Arr[14] := FALSE;
   TL_PIN.Visu_Adv_Arr[15] := FALSE;
   TL_PIN.Visu_Ret_Arr[0] := FALSE;
   TL_PIN.Visu_Ret_Arr[1] := FALSE;
   TL_PIN.Visu_Ret_Arr[2] := FALSE;
   TL_PIN.Visu_Ret_Arr[3] := FALSE;
   TL_PIN.Visu_Ret_Arr[4] := FALSE;
   TL_PIN.Visu_Ret_Arr[5] := FALSE;
   TL_PIN.Visu_Ret_Arr[6] := FALSE;
   TL_PIN.Visu_Ret_Arr[7] := FALSE;
   TL_PIN.Visu_Ret_Arr[8] := FALSE;
   TL_PIN.Visu_Ret_Arr[9] := FALSE;
   TL_PIN.Visu_Ret_Arr[10] := FALSE;
   TL_PIN.Visu_Ret_Arr[11] := FALSE;
   TL_PIN.Visu_Ret_Arr[12] := FALSE;
   TL_PIN.Visu_Ret_Arr[13] := FALSE;
   TL_PIN.Visu_Ret_Arr[14] := FALSE;
   TL_PIN.Visu_Ret_Arr[15] := FALSE;
   TL_PIN.BLK_Move_Ret := 0;
   TL_PIN.Enable := FALSE;
   TL_PIN.Adv_End := FALSE;
   TL_PIN.Ret_End := FALSE;
   LM_BT_CHANGE.General_JIG := FALSE;
   LM_BT_CHANGE.DAECHA_ID_ON := FALSE;
   LM_BT_CHANGE.M_Ready := FALSE;
   LM_BT_CHANGE.SOL_Adv := FALSE;
   LM_BT_CHANGE.SOL_Ret := FALSE;
   LM_BT_CHANGE.Adv_Amount := 0;
   LM_BT_CHANGE.Ret_Amount := 0;
   LM_BT_CHANGE.LS_Adv1 := FALSE;
   LM_BT_CHANGE.LS_Ret1 := FALSE;
   LM_BT_CHANGE.LS_Adv2 := FALSE;
   LM_BT_CHANGE.LS_Ret2 := FALSE;
   LM_BT_CHANGE.LS_Adv3 := FALSE;
   LM_BT_CHANGE.LS_Ret3 := FALSE;
   LM_BT_CHANGE.LS_Adv4 := FALSE;
   LM_BT_CHANGE.LS_Ret4 := FALSE;
   LM_BT_CHANGE.LS_Adv5 := FALSE;
   LM_BT_CHANGE.LS_Ret5 := FALSE;
   LM_BT_CHANGE.LS_Adv6 := FALSE;
   LM_BT_CHANGE.LS_Ret6 := FALSE;
   LM_BT_CHANGE.LS_Adv7 := FALSE;
   LM_BT_CHANGE.LS_Ret7 := FALSE;
   LM_BT_CHANGE.LS_Adv8 := FALSE;
   LM_BT_CHANGE.LS_Ret8 := FALSE;
   LM_BT_CHANGE.LS_Adv9 := FALSE;
   LM_BT_CHANGE.LS_Ret9 := FALSE;
   LM_BT_CHANGE.LS_Adv10 := FALSE;
   LM_BT_CHANGE.LS_Ret10 := FALSE;
   LM_BT_CHANGE.T_CHK1 := T#0MS;
   LM_BT_CHANGE.T_CHK2 := T#0MS;
   LM_BT_CHANGE.PB_Error_Rst := FALSE;
   LM_BT_CHANGE.PB_Lamp_CHK := FALSE;
   LM_BT_CHANGE.M_FLICK := FALSE;
   LM_BT_CHANGE.M_Adv_Err := FALSE;
   LM_BT_CHANGE.M_Ret_Err := FALSE;
   LM_BT_CHANGE.LP_Adv := FALSE;
   LM_BT_CHANGE.LP_Ret := FALSE;
   LM_BT_CHANGE.Visu_Adv := W#16#0;
   LM_BT_CHANGE.Visu_Ret := W#16#0;
   LM_BT_CHANGE.Error_T1.IN := FALSE;
   LM_BT_CHANGE.Error_T1.PT := T#0MS;
   LM_BT_CHANGE.Error_T1.Q := FALSE;
   LM_BT_CHANGE.Error_T1.ET := T#0MS;
   LM_BT_CHANGE.Error_T1.STATE := B#16#0;
   LM_BT_CHANGE.Error_T1.STIME := T#0MS;
   LM_BT_CHANGE.Error_T1.ATIME := T#0MS;
   LM_BT_CHANGE.Error_T2.IN := FALSE;
   LM_BT_CHANGE.Error_T2.PT := T#0MS;
   LM_BT_CHANGE.Error_T2.Q := FALSE;
   LM_BT_CHANGE.Error_T2.ET := T#0MS;
   LM_BT_CHANGE.Error_T2.STATE := B#16#0;
   LM_BT_CHANGE.Error_T2.STIME := T#0MS;
   LM_BT_CHANGE.Error_T2.ATIME := T#0MS;
   LM_BT_CHANGE.Adv_End_Delay.IN := FALSE;
   LM_BT_CHANGE.Adv_End_Delay.PT := T#0MS;
   LM_BT_CHANGE.Adv_End_Delay.Q := FALSE;
   LM_BT_CHANGE.Adv_End_Delay.ET := T#0MS;
   LM_BT_CHANGE.Adv_End_Delay.STATE := B#16#0;
   LM_BT_CHANGE.Adv_End_Delay.STIME := T#0MS;
   LM_BT_CHANGE.Adv_End_Delay.ATIME := T#0MS;
   LM_BT_CHANGE.Ret_End_Delay.IN := FALSE;
   LM_BT_CHANGE.Ret_End_Delay.PT := T#0MS;
   LM_BT_CHANGE.Ret_End_Delay.Q := FALSE;
   LM_BT_CHANGE.Ret_End_Delay.ET := T#0MS;
   LM_BT_CHANGE.Ret_End_Delay.STATE := B#16#0;
   LM_BT_CHANGE.Ret_End_Delay.STIME := T#0MS;
   LM_BT_CHANGE.Ret_End_Delay.ATIME := T#0MS;
   LM_BT_CHANGE.Adv_End_Aux := FALSE;
   LM_BT_CHANGE.Ret_End_Aux := FALSE;
   LM_BT_CHANGE.CHK_Aux1 := FALSE;
   LM_BT_CHANGE.CHK_Aux2 := FALSE;
   LM_BT_CHANGE.Error_T1_DN := FALSE;
   LM_BT_CHANGE.Error_T2_DN := FALSE;
   LM_BT_CHANGE.Adv_Memo := FALSE;
   LM_BT_CHANGE.Visu_Adv_Arr[0] := FALSE;
   LM_BT_CHANGE.Visu_Adv_Arr[1] := FALSE;
   LM_BT_CHANGE.Visu_Adv_Arr[2] := FALSE;
   LM_BT_CHANGE.Visu_Adv_Arr[3] := FALSE;
   LM_BT_CHANGE.Visu_Adv_Arr[4] := FALSE;
   LM_BT_CHANGE.Visu_Adv_Arr[5] := FALSE;
   LM_BT_CHANGE.Visu_Adv_Arr[6] := FALSE;
   LM_BT_CHANGE.Visu_Adv_Arr[7] := FALSE;
   LM_BT_CHANGE.Visu_Adv_Arr[8] := FALSE;
   LM_BT_CHANGE.Visu_Adv_Arr[9] := FALSE;
   LM_BT_CHANGE.Visu_Adv_Arr[10] := FALSE;
   LM_BT_CHANGE.Visu_Adv_Arr[11] := FALSE;
   LM_BT_CHANGE.Visu_Adv_Arr[12] := FALSE;
   LM_BT_CHANGE.Visu_Adv_Arr[13] := FALSE;
   LM_BT_CHANGE.Visu_Adv_Arr[14] := FALSE;
   LM_BT_CHANGE.Visu_Adv_Arr[15] := FALSE;
   LM_BT_CHANGE.Visu_Ret_Arr[0] := FALSE;
   LM_BT_CHANGE.Visu_Ret_Arr[1] := FALSE;
   LM_BT_CHANGE.Visu_Ret_Arr[2] := FALSE;
   LM_BT_CHANGE.Visu_Ret_Arr[3] := FALSE;
   LM_BT_CHANGE.Visu_Ret_Arr[4] := FALSE;
   LM_BT_CHANGE.Visu_Ret_Arr[5] := FALSE;
   LM_BT_CHANGE.Visu_Ret_Arr[6] := FALSE;
   LM_BT_CHANGE.Visu_Ret_Arr[7] := FALSE;
   LM_BT_CHANGE.Visu_Ret_Arr[8] := FALSE;
   LM_BT_CHANGE.Visu_Ret_Arr[9] := FALSE;
   LM_BT_CHANGE.Visu_Ret_Arr[10] := FALSE;
   LM_BT_CHANGE.Visu_Ret_Arr[11] := FALSE;
   LM_BT_CHANGE.Visu_Ret_Arr[12] := FALSE;
   LM_BT_CHANGE.Visu_Ret_Arr[13] := FALSE;
   LM_BT_CHANGE.Visu_Ret_Arr[14] := FALSE;
   LM_BT_CHANGE.Visu_Ret_Arr[15] := FALSE;
   LM_BT_CHANGE.BLK_Move_Ret := 0;
   LM_BT_CHANGE.Enable := FALSE;
   LM_BT_CHANGE.M_Adv_End := FALSE;
   LM_BT_CHANGE.M_Ret_End := FALSE;
   LM_CLAMP.Enable_Aux := FALSE;
   LM_CLAMP.Adv_Amount := 0;
   LM_CLAMP.Ret_Amount := 0;
   LM_CLAMP.LS_Adv1 := FALSE;
   LM_CLAMP.LS_Ret1 := FALSE;
   LM_CLAMP.LS_Adv2 := FALSE;
   LM_CLAMP.LS_Ret2 := FALSE;
   LM_CLAMP.LS_Adv3 := FALSE;
   LM_CLAMP.LS_Ret3 := FALSE;
   LM_CLAMP.LS_Adv4 := FALSE;
   LM_CLAMP.LS_Ret4 := FALSE;
   LM_CLAMP.SOL_Adv := FALSE;
   LM_CLAMP.SOL_Ret := FALSE;
   LM_CLAMP.M_Ready := FALSE;
   LM_CLAMP.T_CHK1 := T#0MS;
   LM_CLAMP.T_CHK2 := T#0MS;
   LM_CLAMP.PB_Lamp_CHK := FALSE;
   LM_CLAMP.PB_Error_Rst := FALSE;
   LM_CLAMP.M_FLICK := FALSE;
   LM_CLAMP.M_Adv_Err := FALSE;
   LM_CLAMP.M_Ret_Err := FALSE;
   LM_CLAMP.LP_Adv := FALSE;
   LM_CLAMP.LP_Ret := FALSE;
   LM_CLAMP.Visu_Adv := W#16#0;
   LM_CLAMP.Visu_Ret := W#16#0;
   LM_CLAMP.Error_T1.IN := FALSE;
   LM_CLAMP.Error_T1.PT := T#0MS;
   LM_CLAMP.Error_T1.Q := FALSE;
   LM_CLAMP.Error_T1.ET := T#0MS;
   LM_CLAMP.Error_T1.STATE := B#16#0;
   LM_CLAMP.Error_T1.STIME := T#0MS;
   LM_CLAMP.Error_T1.ATIME := T#0MS;
   LM_CLAMP.Error_T2.IN := FALSE;
   LM_CLAMP.Error_T2.PT := T#0MS;
   LM_CLAMP.Error_T2.Q := FALSE;
   LM_CLAMP.Error_T2.ET := T#0MS;
   LM_CLAMP.Error_T2.STATE := B#16#0;
   LM_CLAMP.Error_T2.STIME := T#0MS;
   LM_CLAMP.Error_T2.ATIME := T#0MS;
   LM_CLAMP.CHK_Aux1 := FALSE;
   LM_CLAMP.CHK_Aux2 := FALSE;
   LM_CLAMP.Error_T1_DN := FALSE;
   LM_CLAMP.Error_T2_DN := FALSE;
   LM_CLAMP.Adv_Memo := FALSE;
   LM_CLAMP.Visu_Adv_Arr[0] := FALSE;
   LM_CLAMP.Visu_Adv_Arr[1] := FALSE;
   LM_CLAMP.Visu_Adv_Arr[2] := FALSE;
   LM_CLAMP.Visu_Adv_Arr[3] := FALSE;
   LM_CLAMP.Visu_Adv_Arr[4] := FALSE;
   LM_CLAMP.Visu_Adv_Arr[5] := FALSE;
   LM_CLAMP.Visu_Adv_Arr[6] := FALSE;
   LM_CLAMP.Visu_Adv_Arr[7] := FALSE;
   LM_CLAMP.Visu_Adv_Arr[8] := FALSE;
   LM_CLAMP.Visu_Adv_Arr[9] := FALSE;
   LM_CLAMP.Visu_Adv_Arr[10] := FALSE;
   LM_CLAMP.Visu_Adv_Arr[11] := FALSE;
   LM_CLAMP.Visu_Adv_Arr[12] := FALSE;
   LM_CLAMP.Visu_Adv_Arr[13] := FALSE;
   LM_CLAMP.Visu_Adv_Arr[14] := FALSE;
   LM_CLAMP.Visu_Adv_Arr[15] := FALSE;
   LM_CLAMP.Visu_Ret_Arr[0] := FALSE;
   LM_CLAMP.Visu_Ret_Arr[1] := FALSE;
   LM_CLAMP.Visu_Ret_Arr[2] := FALSE;
   LM_CLAMP.Visu_Ret_Arr[3] := FALSE;
   LM_CLAMP.Visu_Ret_Arr[4] := FALSE;
   LM_CLAMP.Visu_Ret_Arr[5] := FALSE;
   LM_CLAMP.Visu_Ret_Arr[6] := FALSE;
   LM_CLAMP.Visu_Ret_Arr[7] := FALSE;
   LM_CLAMP.Visu_Ret_Arr[8] := FALSE;
   LM_CLAMP.Visu_Ret_Arr[9] := FALSE;
   LM_CLAMP.Visu_Ret_Arr[10] := FALSE;
   LM_CLAMP.Visu_Ret_Arr[11] := FALSE;
   LM_CLAMP.Visu_Ret_Arr[12] := FALSE;
   LM_CLAMP.Visu_Ret_Arr[13] := FALSE;
   LM_CLAMP.Visu_Ret_Arr[14] := FALSE;
   LM_CLAMP.Visu_Ret_Arr[15] := FALSE;
   LM_CLAMP.BLK_Move_Ret := 0;
   LM_CLAMP.Enable := FALSE;
   LM_CLAMP.Adv_End := FALSE;
   LM_CLAMP.Ret_End := FALSE;
   LM_PIN.Enable_Aux := FALSE;
   LM_PIN.Adv_Amount := 0;
   LM_PIN.Ret_Amount := 0;
   LM_PIN.LS_Adv1 := FALSE;
   LM_PIN.LS_Ret1 := FALSE;
   LM_PIN.LS_Adv2 := FALSE;
   LM_PIN.LS_Ret2 := FALSE;
   LM_PIN.LS_Adv3 := FALSE;
   LM_PIN.LS_Ret3 := FALSE;
   LM_PIN.LS_Adv4 := FALSE;
   LM_PIN.LS_Ret4 := FALSE;
   LM_PIN.SOL_Adv := FALSE;
   LM_PIN.SOL_Ret := FALSE;
   LM_PIN.M_Ready := FALSE;
   LM_PIN.T_CHK1 := T#0MS;
   LM_PIN.T_CHK2 := T#0MS;
   LM_PIN.PB_Lamp_CHK := FALSE;
   LM_PIN.PB_Error_Rst := FALSE;
   LM_PIN.M_FLICK := FALSE;
   LM_PIN.M_Adv_Err := FALSE;
   LM_PIN.M_Ret_Err := FALSE;
   LM_PIN.LP_Adv := FALSE;
   LM_PIN.LP_Ret := FALSE;
   LM_PIN.Visu_Adv := W#16#0;
   LM_PIN.Visu_Ret := W#16#0;
   LM_PIN.Error_T1.IN := FALSE;
   LM_PIN.Error_T1.PT := T#0MS;
   LM_PIN.Error_T1.Q := FALSE;
   LM_PIN.Error_T1.ET := T#0MS;
   LM_PIN.Error_T1.STATE := B#16#0;
   LM_PIN.Error_T1.STIME := T#0MS;
   LM_PIN.Error_T1.ATIME := T#0MS;
   LM_PIN.Error_T2.IN := FALSE;
   LM_PIN.Error_T2.PT := T#0MS;
   LM_PIN.Error_T2.Q := FALSE;
   LM_PIN.Error_T2.ET := T#0MS;
   LM_PIN.Error_T2.STATE := B#16#0;
   LM_PIN.Error_T2.STIME := T#0MS;
   LM_PIN.Error_T2.ATIME := T#0MS;
   LM_PIN.CHK_Aux1 := FALSE;
   LM_PIN.CHK_Aux2 := FALSE;
   LM_PIN.Error_T1_DN := FALSE;
   LM_PIN.Error_T2_DN := FALSE;
   LM_PIN.Adv_Memo := FALSE;
   LM_PIN.Visu_Adv_Arr[0] := FALSE;
   LM_PIN.Visu_Adv_Arr[1] := FALSE;
   LM_PIN.Visu_Adv_Arr[2] := FALSE;
   LM_PIN.Visu_Adv_Arr[3] := FALSE;
   LM_PIN.Visu_Adv_Arr[4] := FALSE;
   LM_PIN.Visu_Adv_Arr[5] := FALSE;
   LM_PIN.Visu_Adv_Arr[6] := FALSE;
   LM_PIN.Visu_Adv_Arr[7] := FALSE;
   LM_PIN.Visu_Adv_Arr[8] := FALSE;
   LM_PIN.Visu_Adv_Arr[9] := FALSE;
   LM_PIN.Visu_Adv_Arr[10] := FALSE;
   LM_PIN.Visu_Adv_Arr[11] := FALSE;
   LM_PIN.Visu_Adv_Arr[12] := FALSE;
   LM_PIN.Visu_Adv_Arr[13] := FALSE;
   LM_PIN.Visu_Adv_Arr[14] := FALSE;
   LM_PIN.Visu_Adv_Arr[15] := FALSE;
   LM_PIN.Visu_Ret_Arr[0] := FALSE;
   LM_PIN.Visu_Ret_Arr[1] := FALSE;
   LM_PIN.Visu_Ret_Arr[2] := FALSE;
   LM_PIN.Visu_Ret_Arr[3] := FALSE;
   LM_PIN.Visu_Ret_Arr[4] := FALSE;
   LM_PIN.Visu_Ret_Arr[5] := FALSE;
   LM_PIN.Visu_Ret_Arr[6] := FALSE;
   LM_PIN.Visu_Ret_Arr[7] := FALSE;
   LM_PIN.Visu_Ret_Arr[8] := FALSE;
   LM_PIN.Visu_Ret_Arr[9] := FALSE;
   LM_PIN.Visu_Ret_Arr[10] := FALSE;
   LM_PIN.Visu_Ret_Arr[11] := FALSE;
   LM_PIN.Visu_Ret_Arr[12] := FALSE;
   LM_PIN.Visu_Ret_Arr[13] := FALSE;
   LM_PIN.Visu_Ret_Arr[14] := FALSE;
   LM_PIN.Visu_Ret_Arr[15] := FALSE;
   LM_PIN.BLK_Move_Ret := 0;
   LM_PIN.Enable := FALSE;
   LM_PIN.Adv_End := FALSE;
   LM_PIN.Ret_End := FALSE;
   LM_INDEX_CLAMP.Enable_Aux := FALSE;
   LM_INDEX_CLAMP.Adv_Amount := 0;
   LM_INDEX_CLAMP.Ret_Amount := 0;
   LM_INDEX_CLAMP.LS_Adv1 := FALSE;
   LM_INDEX_CLAMP.LS_Ret1 := FALSE;
   LM_INDEX_CLAMP.LS_Adv2 := FALSE;
   LM_INDEX_CLAMP.LS_Ret2 := FALSE;
   LM_INDEX_CLAMP.LS_Adv3 := FALSE;
   LM_INDEX_CLAMP.LS_Ret3 := FALSE;
   LM_INDEX_CLAMP.LS_Adv4 := FALSE;
   LM_INDEX_CLAMP.LS_Ret4 := FALSE;
   LM_INDEX_CLAMP.SOL_Adv := FALSE;
   LM_INDEX_CLAMP.SOL_Ret := FALSE;
   LM_INDEX_CLAMP.M_Ready := FALSE;
   LM_INDEX_CLAMP.T_CHK1 := T#0MS;
   LM_INDEX_CLAMP.T_CHK2 := T#0MS;
   LM_INDEX_CLAMP.PB_Lamp_CHK := FALSE;
   LM_INDEX_CLAMP.PB_Error_Rst := FALSE;
   LM_INDEX_CLAMP.M_FLICK := FALSE;
   LM_INDEX_CLAMP.M_Adv_Err := FALSE;
   LM_INDEX_CLAMP.M_Ret_Err := FALSE;
   LM_INDEX_CLAMP.LP_Adv := FALSE;
   LM_INDEX_CLAMP.LP_Ret := FALSE;
   LM_INDEX_CLAMP.Visu_Adv := W#16#0;
   LM_INDEX_CLAMP.Visu_Ret := W#16#0;
   LM_INDEX_CLAMP.Error_T1.IN := FALSE;
   LM_INDEX_CLAMP.Error_T1.PT := T#0MS;
   LM_INDEX_CLAMP.Error_T1.Q := FALSE;
   LM_INDEX_CLAMP.Error_T1.ET := T#0MS;
   LM_INDEX_CLAMP.Error_T1.STATE := B#16#0;
   LM_INDEX_CLAMP.Error_T1.STIME := T#0MS;
   LM_INDEX_CLAMP.Error_T1.ATIME := T#0MS;
   LM_INDEX_CLAMP.Error_T2.IN := FALSE;
   LM_INDEX_CLAMP.Error_T2.PT := T#0MS;
   LM_INDEX_CLAMP.Error_T2.Q := FALSE;
   LM_INDEX_CLAMP.Error_T2.ET := T#0MS;
   LM_INDEX_CLAMP.Error_T2.STATE := B#16#0;
   LM_INDEX_CLAMP.Error_T2.STIME := T#0MS;
   LM_INDEX_CLAMP.Error_T2.ATIME := T#0MS;
   LM_INDEX_CLAMP.CHK_Aux1 := FALSE;
   LM_INDEX_CLAMP.CHK_Aux2 := FALSE;
   LM_INDEX_CLAMP.Error_T1_DN := FALSE;
   LM_INDEX_CLAMP.Error_T2_DN := FALSE;
   LM_INDEX_CLAMP.Adv_Memo := FALSE;
   LM_INDEX_CLAMP.Visu_Adv_Arr[0] := FALSE;
   LM_INDEX_CLAMP.Visu_Adv_Arr[1] := FALSE;
   LM_INDEX_CLAMP.Visu_Adv_Arr[2] := FALSE;
   LM_INDEX_CLAMP.Visu_Adv_Arr[3] := FALSE;
   LM_INDEX_CLAMP.Visu_Adv_Arr[4] := FALSE;
   LM_INDEX_CLAMP.Visu_Adv_Arr[5] := FALSE;
   LM_INDEX_CLAMP.Visu_Adv_Arr[6] := FALSE;
   LM_INDEX_CLAMP.Visu_Adv_Arr[7] := FALSE;
   LM_INDEX_CLAMP.Visu_Adv_Arr[8] := FALSE;
   LM_INDEX_CLAMP.Visu_Adv_Arr[9] := FALSE;
   LM_INDEX_CLAMP.Visu_Adv_Arr[10] := FALSE;
   LM_INDEX_CLAMP.Visu_Adv_Arr[11] := FALSE;
   LM_INDEX_CLAMP.Visu_Adv_Arr[12] := FALSE;
   LM_INDEX_CLAMP.Visu_Adv_Arr[13] := FALSE;
   LM_INDEX_CLAMP.Visu_Adv_Arr[14] := FALSE;
   LM_INDEX_CLAMP.Visu_Adv_Arr[15] := FALSE;
   LM_INDEX_CLAMP.Visu_Ret_Arr[0] := FALSE;
   LM_INDEX_CLAMP.Visu_Ret_Arr[1] := FALSE;
   LM_INDEX_CLAMP.Visu_Ret_Arr[2] := FALSE;
   LM_INDEX_CLAMP.Visu_Ret_Arr[3] := FALSE;
   LM_INDEX_CLAMP.Visu_Ret_Arr[4] := FALSE;
   LM_INDEX_CLAMP.Visu_Ret_Arr[5] := FALSE;
   LM_INDEX_CLAMP.Visu_Ret_Arr[6] := FALSE;
   LM_INDEX_CLAMP.Visu_Ret_Arr[7] := FALSE;
   LM_INDEX_CLAMP.Visu_Ret_Arr[8] := FALSE;
   LM_INDEX_CLAMP.Visu_Ret_Arr[9] := FALSE;
   LM_INDEX_CLAMP.Visu_Ret_Arr[10] := FALSE;
   LM_INDEX_CLAMP.Visu_Ret_Arr[11] := FALSE;
   LM_INDEX_CLAMP.Visu_Ret_Arr[12] := FALSE;
   LM_INDEX_CLAMP.Visu_Ret_Arr[13] := FALSE;
   LM_INDEX_CLAMP.Visu_Ret_Arr[14] := FALSE;
   LM_INDEX_CLAMP.Visu_Ret_Arr[15] := FALSE;
   LM_INDEX_CLAMP.BLK_Move_Ret := 0;
   LM_INDEX_CLAMP.Enable := FALSE;
   LM_INDEX_CLAMP.Adv_End := FALSE;
   LM_INDEX_CLAMP.Ret_End := FALSE;
   LM_INDEX_PIN.Enable_Aux := FALSE;
   LM_INDEX_PIN.Adv_Amount := 0;
   LM_INDEX_PIN.Ret_Amount := 0;
   LM_INDEX_PIN.LS_Adv1 := FALSE;
   LM_INDEX_PIN.LS_Ret1 := FALSE;
   LM_INDEX_PIN.LS_Adv2 := FALSE;
   LM_INDEX_PIN.LS_Ret2 := FALSE;
   LM_INDEX_PIN.LS_Adv3 := FALSE;
   LM_INDEX_PIN.LS_Ret3 := FALSE;
   LM_INDEX_PIN.LS_Adv4 := FALSE;
   LM_INDEX_PIN.LS_Ret4 := FALSE;
   LM_INDEX_PIN.SOL_Adv := FALSE;
   LM_INDEX_PIN.SOL_Ret := FALSE;
   LM_INDEX_PIN.M_Ready := FALSE;
   LM_INDEX_PIN.T_CHK1 := T#0MS;
   LM_INDEX_PIN.T_CHK2 := T#0MS;
   LM_INDEX_PIN.PB_Lamp_CHK := FALSE;
   LM_INDEX_PIN.PB_Error_Rst := FALSE;
   LM_INDEX_PIN.M_FLICK := FALSE;
   LM_INDEX_PIN.M_Adv_Err := FALSE;
   LM_INDEX_PIN.M_Ret_Err := FALSE;
   LM_INDEX_PIN.LP_Adv := FALSE;
   LM_INDEX_PIN.LP_Ret := FALSE;
   LM_INDEX_PIN.Visu_Adv := W#16#0;
   LM_INDEX_PIN.Visu_Ret := W#16#0;
   LM_INDEX_PIN.Error_T1.IN := FALSE;
   LM_INDEX_PIN.Error_T1.PT := T#0MS;
   LM_INDEX_PIN.Error_T1.Q := FALSE;
   LM_INDEX_PIN.Error_T1.ET := T#0MS;
   LM_INDEX_PIN.Error_T1.STATE := B#16#0;
   LM_INDEX_PIN.Error_T1.STIME := T#0MS;
   LM_INDEX_PIN.Error_T1.ATIME := T#0MS;
   LM_INDEX_PIN.Error_T2.IN := FALSE;
   LM_INDEX_PIN.Error_T2.PT := T#0MS;
   LM_INDEX_PIN.Error_T2.Q := FALSE;
   LM_INDEX_PIN.Error_T2.ET := T#0MS;
   LM_INDEX_PIN.Error_T2.STATE := B#16#0;
   LM_INDEX_PIN.Error_T2.STIME := T#0MS;
   LM_INDEX_PIN.Error_T2.ATIME := T#0MS;
   LM_INDEX_PIN.CHK_Aux1 := FALSE;
   LM_INDEX_PIN.CHK_Aux2 := FALSE;
   LM_INDEX_PIN.Error_T1_DN := FALSE;
   LM_INDEX_PIN.Error_T2_DN := FALSE;
   LM_INDEX_PIN.Adv_Memo := FALSE;
   LM_INDEX_PIN.Visu_Adv_Arr[0] := FALSE;
   LM_INDEX_PIN.Visu_Adv_Arr[1] := FALSE;
   LM_INDEX_PIN.Visu_Adv_Arr[2] := FALSE;
   LM_INDEX_PIN.Visu_Adv_Arr[3] := FALSE;
   LM_INDEX_PIN.Visu_Adv_Arr[4] := FALSE;
   LM_INDEX_PIN.Visu_Adv_Arr[5] := FALSE;
   LM_INDEX_PIN.Visu_Adv_Arr[6] := FALSE;
   LM_INDEX_PIN.Visu_Adv_Arr[7] := FALSE;
   LM_INDEX_PIN.Visu_Adv_Arr[8] := FALSE;
   LM_INDEX_PIN.Visu_Adv_Arr[9] := FALSE;
   LM_INDEX_PIN.Visu_Adv_Arr[10] := FALSE;
   LM_INDEX_PIN.Visu_Adv_Arr[11] := FALSE;
   LM_INDEX_PIN.Visu_Adv_Arr[12] := FALSE;
   LM_INDEX_PIN.Visu_Adv_Arr[13] := FALSE;
   LM_INDEX_PIN.Visu_Adv_Arr[14] := FALSE;
   LM_INDEX_PIN.Visu_Adv_Arr[15] := FALSE;
   LM_INDEX_PIN.Visu_Ret_Arr[0] := FALSE;
   LM_INDEX_PIN.Visu_Ret_Arr[1] := FALSE;
   LM_INDEX_PIN.Visu_Ret_Arr[2] := FALSE;
   LM_INDEX_PIN.Visu_Ret_Arr[3] := FALSE;
   LM_INDEX_PIN.Visu_Ret_Arr[4] := FALSE;
   LM_INDEX_PIN.Visu_Ret_Arr[5] := FALSE;
   LM_INDEX_PIN.Visu_Ret_Arr[6] := FALSE;
   LM_INDEX_PIN.Visu_Ret_Arr[7] := FALSE;
   LM_INDEX_PIN.Visu_Ret_Arr[8] := FALSE;
   LM_INDEX_PIN.Visu_Ret_Arr[9] := FALSE;
   LM_INDEX_PIN.Visu_Ret_Arr[10] := FALSE;
   LM_INDEX_PIN.Visu_Ret_Arr[11] := FALSE;
   LM_INDEX_PIN.Visu_Ret_Arr[12] := FALSE;
   LM_INDEX_PIN.Visu_Ret_Arr[13] := FALSE;
   LM_INDEX_PIN.Visu_Ret_Arr[14] := FALSE;
   LM_INDEX_PIN.Visu_Ret_Arr[15] := FALSE;
   LM_INDEX_PIN.BLK_Move_Ret := 0;
   LM_INDEX_PIN.Enable := FALSE;
   LM_INDEX_PIN.Adv_End := FALSE;
   LM_INDEX_PIN.Ret_End := FALSE;
   INR_PLT3_UP_DOWN.Enable_Aux := FALSE;
   INR_PLT3_UP_DOWN.Adv_Amount := 0;
   INR_PLT3_UP_DOWN.Ret_Amount := 0;
   INR_PLT3_UP_DOWN.LS_Adv1 := FALSE;
   INR_PLT3_UP_DOWN.LS_Ret1 := FALSE;
   INR_PLT3_UP_DOWN.LS_Adv2 := FALSE;
   INR_PLT3_UP_DOWN.LS_Ret2 := FALSE;
   INR_PLT3_UP_DOWN.LS_Adv3 := FALSE;
   INR_PLT3_UP_DOWN.LS_Ret3 := FALSE;
   INR_PLT3_UP_DOWN.LS_Adv4 := FALSE;
   INR_PLT3_UP_DOWN.LS_Ret4 := FALSE;
   INR_PLT3_UP_DOWN.SOL_Adv := FALSE;
   INR_PLT3_UP_DOWN.SOL_Ret := FALSE;
   INR_PLT3_UP_DOWN.M_Ready := FALSE;
   INR_PLT3_UP_DOWN.T_CHK1 := T#0MS;
   INR_PLT3_UP_DOWN.T_CHK2 := T#0MS;
   INR_PLT3_UP_DOWN.PB_Lamp_CHK := FALSE;
   INR_PLT3_UP_DOWN.PB_Error_Rst := FALSE;
   INR_PLT3_UP_DOWN.M_FLICK := FALSE;
   INR_PLT3_UP_DOWN.M_Adv_Err := FALSE;
   INR_PLT3_UP_DOWN.M_Ret_Err := FALSE;
   INR_PLT3_UP_DOWN.LP_Adv := FALSE;
   INR_PLT3_UP_DOWN.LP_Ret := FALSE;
   INR_PLT3_UP_DOWN.Visu_Adv := W#16#0;
   INR_PLT3_UP_DOWN.Visu_Ret := W#16#0;
   INR_PLT3_UP_DOWN.Error_T1.IN := FALSE;
   INR_PLT3_UP_DOWN.Error_T1.PT := T#0MS;
   INR_PLT3_UP_DOWN.Error_T1.Q := FALSE;
   INR_PLT3_UP_DOWN.Error_T1.ET := T#0MS;
   INR_PLT3_UP_DOWN.Error_T1.STATE := B#16#0;
   INR_PLT3_UP_DOWN.Error_T1.STIME := T#0MS;
   INR_PLT3_UP_DOWN.Error_T1.ATIME := T#0MS;
   INR_PLT3_UP_DOWN.Error_T2.IN := FALSE;
   INR_PLT3_UP_DOWN.Error_T2.PT := T#0MS;
   INR_PLT3_UP_DOWN.Error_T2.Q := FALSE;
   INR_PLT3_UP_DOWN.Error_T2.ET := T#0MS;
   INR_PLT3_UP_DOWN.Error_T2.STATE := B#16#0;
   INR_PLT3_UP_DOWN.Error_T2.STIME := T#0MS;
   INR_PLT3_UP_DOWN.Error_T2.ATIME := T#0MS;
   INR_PLT3_UP_DOWN.CHK_Aux1 := FALSE;
   INR_PLT3_UP_DOWN.CHK_Aux2 := FALSE;
   INR_PLT3_UP_DOWN.Error_T1_DN := FALSE;
   INR_PLT3_UP_DOWN.Error_T2_DN := FALSE;
   INR_PLT3_UP_DOWN.Adv_Memo := FALSE;
   INR_PLT3_UP_DOWN.Visu_Adv_Arr[0] := FALSE;
   INR_PLT3_UP_DOWN.Visu_Adv_Arr[1] := FALSE;
   INR_PLT3_UP_DOWN.Visu_Adv_Arr[2] := FALSE;
   INR_PLT3_UP_DOWN.Visu_Adv_Arr[3] := FALSE;
   INR_PLT3_UP_DOWN.Visu_Adv_Arr[4] := FALSE;
   INR_PLT3_UP_DOWN.Visu_Adv_Arr[5] := FALSE;
   INR_PLT3_UP_DOWN.Visu_Adv_Arr[6] := FALSE;
   INR_PLT3_UP_DOWN.Visu_Adv_Arr[7] := FALSE;
   INR_PLT3_UP_DOWN.Visu_Adv_Arr[8] := FALSE;
   INR_PLT3_UP_DOWN.Visu_Adv_Arr[9] := FALSE;
   INR_PLT3_UP_DOWN.Visu_Adv_Arr[10] := FALSE;
   INR_PLT3_UP_DOWN.Visu_Adv_Arr[11] := FALSE;
   INR_PLT3_UP_DOWN.Visu_Adv_Arr[12] := FALSE;
   INR_PLT3_UP_DOWN.Visu_Adv_Arr[13] := FALSE;
   INR_PLT3_UP_DOWN.Visu_Adv_Arr[14] := FALSE;
   INR_PLT3_UP_DOWN.Visu_Adv_Arr[15] := FALSE;
   INR_PLT3_UP_DOWN.Visu_Ret_Arr[0] := FALSE;
   INR_PLT3_UP_DOWN.Visu_Ret_Arr[1] := FALSE;
   INR_PLT3_UP_DOWN.Visu_Ret_Arr[2] := FALSE;
   INR_PLT3_UP_DOWN.Visu_Ret_Arr[3] := FALSE;
   INR_PLT3_UP_DOWN.Visu_Ret_Arr[4] := FALSE;
   INR_PLT3_UP_DOWN.Visu_Ret_Arr[5] := FALSE;
   INR_PLT3_UP_DOWN.Visu_Ret_Arr[6] := FALSE;
   INR_PLT3_UP_DOWN.Visu_Ret_Arr[7] := FALSE;
   INR_PLT3_UP_DOWN.Visu_Ret_Arr[8] := FALSE;
   INR_PLT3_UP_DOWN.Visu_Ret_Arr[9] := FALSE;
   INR_PLT3_UP_DOWN.Visu_Ret_Arr[10] := FALSE;
   INR_PLT3_UP_DOWN.Visu_Ret_Arr[11] := FALSE;
   INR_PLT3_UP_DOWN.Visu_Ret_Arr[12] := FALSE;
   INR_PLT3_UP_DOWN.Visu_Ret_Arr[13] := FALSE;
   INR_PLT3_UP_DOWN.Visu_Ret_Arr[14] := FALSE;
   INR_PLT3_UP_DOWN.Visu_Ret_Arr[15] := FALSE;
   INR_PLT3_UP_DOWN.BLK_Move_Ret := 0;
   INR_PLT3_UP_DOWN.Enable := FALSE;
   INR_PLT3_UP_DOWN.Adv_End := FALSE;
   INR_PLT3_UP_DOWN.Ret_End := FALSE;
   INR_PLT3_LOCK.Enable_Aux := FALSE;
   INR_PLT3_LOCK.Adv_Amount := 0;
   INR_PLT3_LOCK.Ret_Amount := 0;
   INR_PLT3_LOCK.LS_Adv1 := FALSE;
   INR_PLT3_LOCK.LS_Ret1 := FALSE;
   INR_PLT3_LOCK.LS_Adv2 := FALSE;
   INR_PLT3_LOCK.LS_Ret2 := FALSE;
   INR_PLT3_LOCK.LS_Adv3 := FALSE;
   INR_PLT3_LOCK.LS_Ret3 := FALSE;
   INR_PLT3_LOCK.LS_Adv4 := FALSE;
   INR_PLT3_LOCK.LS_Ret4 := FALSE;
   INR_PLT3_LOCK.SOL_Adv := FALSE;
   INR_PLT3_LOCK.SOL_Ret := FALSE;
   INR_PLT3_LOCK.M_Ready := FALSE;
   INR_PLT3_LOCK.T_CHK1 := T#0MS;
   INR_PLT3_LOCK.T_CHK2 := T#0MS;
   INR_PLT3_LOCK.PB_Lamp_CHK := FALSE;
   INR_PLT3_LOCK.PB_Error_Rst := FALSE;
   INR_PLT3_LOCK.M_FLICK := FALSE;
   INR_PLT3_LOCK.M_Adv_Err := FALSE;
   INR_PLT3_LOCK.M_Ret_Err := FALSE;
   INR_PLT3_LOCK.LP_Adv := FALSE;
   INR_PLT3_LOCK.LP_Ret := FALSE;
   INR_PLT3_LOCK.Visu_Adv := W#16#0;
   INR_PLT3_LOCK.Visu_Ret := W#16#0;
   INR_PLT3_LOCK.Error_T1.IN := FALSE;
   INR_PLT3_LOCK.Error_T1.PT := T#0MS;
   INR_PLT3_LOCK.Error_T1.Q := FALSE;
   INR_PLT3_LOCK.Error_T1.ET := T#0MS;
   INR_PLT3_LOCK.Error_T1.STATE := B#16#0;
   INR_PLT3_LOCK.Error_T1.STIME := T#0MS;
   INR_PLT3_LOCK.Error_T1.ATIME := T#0MS;
   INR_PLT3_LOCK.Error_T2.IN := FALSE;
   INR_PLT3_LOCK.Error_T2.PT := T#0MS;
   INR_PLT3_LOCK.Error_T2.Q := FALSE;
   INR_PLT3_LOCK.Error_T2.ET := T#0MS;
   INR_PLT3_LOCK.Error_T2.STATE := B#16#0;
   INR_PLT3_LOCK.Error_T2.STIME := T#0MS;
   INR_PLT3_LOCK.Error_T2.ATIME := T#0MS;
   INR_PLT3_LOCK.CHK_Aux1 := FALSE;
   INR_PLT3_LOCK.CHK_Aux2 := FALSE;
   INR_PLT3_LOCK.Error_T1_DN := FALSE;
   INR_PLT3_LOCK.Error_T2_DN := FALSE;
   INR_PLT3_LOCK.Adv_Memo := FALSE;
   INR_PLT3_LOCK.Visu_Adv_Arr[0] := FALSE;
   INR_PLT3_LOCK.Visu_Adv_Arr[1] := FALSE;
   INR_PLT3_LOCK.Visu_Adv_Arr[2] := FALSE;
   INR_PLT3_LOCK.Visu_Adv_Arr[3] := FALSE;
   INR_PLT3_LOCK.Visu_Adv_Arr[4] := FALSE;
   INR_PLT3_LOCK.Visu_Adv_Arr[5] := FALSE;
   INR_PLT3_LOCK.Visu_Adv_Arr[6] := FALSE;
   INR_PLT3_LOCK.Visu_Adv_Arr[7] := FALSE;
   INR_PLT3_LOCK.Visu_Adv_Arr[8] := FALSE;
   INR_PLT3_LOCK.Visu_Adv_Arr[9] := FALSE;
   INR_PLT3_LOCK.Visu_Adv_Arr[10] := FALSE;
   INR_PLT3_LOCK.Visu_Adv_Arr[11] := FALSE;
   INR_PLT3_LOCK.Visu_Adv_Arr[12] := FALSE;
   INR_PLT3_LOCK.Visu_Adv_Arr[13] := FALSE;
   INR_PLT3_LOCK.Visu_Adv_Arr[14] := FALSE;
   INR_PLT3_LOCK.Visu_Adv_Arr[15] := FALSE;
   INR_PLT3_LOCK.Visu_Ret_Arr[0] := FALSE;
   INR_PLT3_LOCK.Visu_Ret_Arr[1] := FALSE;
   INR_PLT3_LOCK.Visu_Ret_Arr[2] := FALSE;
   INR_PLT3_LOCK.Visu_Ret_Arr[3] := FALSE;
   INR_PLT3_LOCK.Visu_Ret_Arr[4] := FALSE;
   INR_PLT3_LOCK.Visu_Ret_Arr[5] := FALSE;
   INR_PLT3_LOCK.Visu_Ret_Arr[6] := FALSE;
   INR_PLT3_LOCK.Visu_Ret_Arr[7] := FALSE;
   INR_PLT3_LOCK.Visu_Ret_Arr[8] := FALSE;
   INR_PLT3_LOCK.Visu_Ret_Arr[9] := FALSE;
   INR_PLT3_LOCK.Visu_Ret_Arr[10] := FALSE;
   INR_PLT3_LOCK.Visu_Ret_Arr[11] := FALSE;
   INR_PLT3_LOCK.Visu_Ret_Arr[12] := FALSE;
   INR_PLT3_LOCK.Visu_Ret_Arr[13] := FALSE;
   INR_PLT3_LOCK.Visu_Ret_Arr[14] := FALSE;
   INR_PLT3_LOCK.Visu_Ret_Arr[15] := FALSE;
   INR_PLT3_LOCK.BLK_Move_Ret := 0;
   INR_PLT3_LOCK.Enable := FALSE;
   INR_PLT3_LOCK.Adv_End := FALSE;
   INR_PLT3_LOCK.Ret_End := FALSE;
   INR_PLT4_UP_DOWN.Enable_Aux := FALSE;
   INR_PLT4_UP_DOWN.Adv_Amount := 0;
   INR_PLT4_UP_DOWN.Ret_Amount := 0;
   INR_PLT4_UP_DOWN.LS_Adv1 := FALSE;
   INR_PLT4_UP_DOWN.LS_Ret1 := FALSE;
   INR_PLT4_UP_DOWN.LS_Adv2 := FALSE;
   INR_PLT4_UP_DOWN.LS_Ret2 := FALSE;
   INR_PLT4_UP_DOWN.LS_Adv3 := FALSE;
   INR_PLT4_UP_DOWN.LS_Ret3 := FALSE;
   INR_PLT4_UP_DOWN.LS_Adv4 := FALSE;
   INR_PLT4_UP_DOWN.LS_Ret4 := FALSE;
   INR_PLT4_UP_DOWN.SOL_Adv := FALSE;
   INR_PLT4_UP_DOWN.SOL_Ret := FALSE;
   INR_PLT4_UP_DOWN.M_Ready := FALSE;
   INR_PLT4_UP_DOWN.T_CHK1 := T#0MS;
   INR_PLT4_UP_DOWN.T_CHK2 := T#0MS;
   INR_PLT4_UP_DOWN.PB_Lamp_CHK := FALSE;
   INR_PLT4_UP_DOWN.PB_Error_Rst := FALSE;
   INR_PLT4_UP_DOWN.M_FLICK := FALSE;
   INR_PLT4_UP_DOWN.M_Adv_Err := FALSE;
   INR_PLT4_UP_DOWN.M_Ret_Err := FALSE;
   INR_PLT4_UP_DOWN.LP_Adv := FALSE;
   INR_PLT4_UP_DOWN.LP_Ret := FALSE;
   INR_PLT4_UP_DOWN.Visu_Adv := W#16#0;
   INR_PLT4_UP_DOWN.Visu_Ret := W#16#0;
   INR_PLT4_UP_DOWN.Error_T1.IN := FALSE;
   INR_PLT4_UP_DOWN.Error_T1.PT := T#0MS;
   INR_PLT4_UP_DOWN.Error_T1.Q := FALSE;
   INR_PLT4_UP_DOWN.Error_T1.ET := T#0MS;
   INR_PLT4_UP_DOWN.Error_T1.STATE := B#16#0;
   INR_PLT4_UP_DOWN.Error_T1.STIME := T#0MS;
   INR_PLT4_UP_DOWN.Error_T1.ATIME := T#0MS;
   INR_PLT4_UP_DOWN.Error_T2.IN := FALSE;
   INR_PLT4_UP_DOWN.Error_T2.PT := T#0MS;
   INR_PLT4_UP_DOWN.Error_T2.Q := FALSE;
   INR_PLT4_UP_DOWN.Error_T2.ET := T#0MS;
   INR_PLT4_UP_DOWN.Error_T2.STATE := B#16#0;
   INR_PLT4_UP_DOWN.Error_T2.STIME := T#0MS;
   INR_PLT4_UP_DOWN.Error_T2.ATIME := T#0MS;
   INR_PLT4_UP_DOWN.CHK_Aux1 := FALSE;
   INR_PLT4_UP_DOWN.CHK_Aux2 := FALSE;
   INR_PLT4_UP_DOWN.Error_T1_DN := FALSE;
   INR_PLT4_UP_DOWN.Error_T2_DN := FALSE;
   INR_PLT4_UP_DOWN.Adv_Memo := FALSE;
   INR_PLT4_UP_DOWN.Visu_Adv_Arr[0] := FALSE;
   INR_PLT4_UP_DOWN.Visu_Adv_Arr[1] := FALSE;
   INR_PLT4_UP_DOWN.Visu_Adv_Arr[2] := FALSE;
   INR_PLT4_UP_DOWN.Visu_Adv_Arr[3] := FALSE;
   INR_PLT4_UP_DOWN.Visu_Adv_Arr[4] := FALSE;
   INR_PLT4_UP_DOWN.Visu_Adv_Arr[5] := FALSE;
   INR_PLT4_UP_DOWN.Visu_Adv_Arr[6] := FALSE;
   INR_PLT4_UP_DOWN.Visu_Adv_Arr[7] := FALSE;
   INR_PLT4_UP_DOWN.Visu_Adv_Arr[8] := FALSE;
   INR_PLT4_UP_DOWN.Visu_Adv_Arr[9] := FALSE;
   INR_PLT4_UP_DOWN.Visu_Adv_Arr[10] := FALSE;
   INR_PLT4_UP_DOWN.Visu_Adv_Arr[11] := FALSE;
   INR_PLT4_UP_DOWN.Visu_Adv_Arr[12] := FALSE;
   INR_PLT4_UP_DOWN.Visu_Adv_Arr[13] := FALSE;
   INR_PLT4_UP_DOWN.Visu_Adv_Arr[14] := FALSE;
   INR_PLT4_UP_DOWN.Visu_Adv_Arr[15] := FALSE;
   INR_PLT4_UP_DOWN.Visu_Ret_Arr[0] := FALSE;
   INR_PLT4_UP_DOWN.Visu_Ret_Arr[1] := FALSE;
   INR_PLT4_UP_DOWN.Visu_Ret_Arr[2] := FALSE;
   INR_PLT4_UP_DOWN.Visu_Ret_Arr[3] := FALSE;
   INR_PLT4_UP_DOWN.Visu_Ret_Arr[4] := FALSE;
   INR_PLT4_UP_DOWN.Visu_Ret_Arr[5] := FALSE;
   INR_PLT4_UP_DOWN.Visu_Ret_Arr[6] := FALSE;
   INR_PLT4_UP_DOWN.Visu_Ret_Arr[7] := FALSE;
   INR_PLT4_UP_DOWN.Visu_Ret_Arr[8] := FALSE;
   INR_PLT4_UP_DOWN.Visu_Ret_Arr[9] := FALSE;
   INR_PLT4_UP_DOWN.Visu_Ret_Arr[10] := FALSE;
   INR_PLT4_UP_DOWN.Visu_Ret_Arr[11] := FALSE;
   INR_PLT4_UP_DOWN.Visu_Ret_Arr[12] := FALSE;
   INR_PLT4_UP_DOWN.Visu_Ret_Arr[13] := FALSE;
   INR_PLT4_UP_DOWN.Visu_Ret_Arr[14] := FALSE;
   INR_PLT4_UP_DOWN.Visu_Ret_Arr[15] := FALSE;
   INR_PLT4_UP_DOWN.BLK_Move_Ret := 0;
   INR_PLT4_UP_DOWN.Enable := FALSE;
   INR_PLT4_UP_DOWN.Adv_End := FALSE;
   INR_PLT4_UP_DOWN.Ret_End := FALSE;
   INR_PLT4_LOCK.Enable_Aux := FALSE;
   INR_PLT4_LOCK.Adv_Amount := 0;
   INR_PLT4_LOCK.Ret_Amount := 0;
   INR_PLT4_LOCK.LS_Adv1 := FALSE;
   INR_PLT4_LOCK.LS_Ret1 := FALSE;
   INR_PLT4_LOCK.LS_Adv2 := FALSE;
   INR_PLT4_LOCK.LS_Ret2 := FALSE;
   INR_PLT4_LOCK.LS_Adv3 := FALSE;
   INR_PLT4_LOCK.LS_Ret3 := FALSE;
   INR_PLT4_LOCK.LS_Adv4 := FALSE;
   INR_PLT4_LOCK.LS_Ret4 := FALSE;
   INR_PLT4_LOCK.SOL_Adv := FALSE;
   INR_PLT4_LOCK.SOL_Ret := FALSE;
   INR_PLT4_LOCK.M_Ready := FALSE;
   INR_PLT4_LOCK.T_CHK1 := T#0MS;
   INR_PLT4_LOCK.T_CHK2 := T#0MS;
   INR_PLT4_LOCK.PB_Lamp_CHK := FALSE;
   INR_PLT4_LOCK.PB_Error_Rst := FALSE;
   INR_PLT4_LOCK.M_FLICK := FALSE;
   INR_PLT4_LOCK.M_Adv_Err := FALSE;
   INR_PLT4_LOCK.M_Ret_Err := FALSE;
   INR_PLT4_LOCK.LP_Adv := FALSE;
   INR_PLT4_LOCK.LP_Ret := FALSE;
   INR_PLT4_LOCK.Visu_Adv := W#16#0;
   INR_PLT4_LOCK.Visu_Ret := W#16#0;
   INR_PLT4_LOCK.Error_T1.IN := FALSE;
   INR_PLT4_LOCK.Error_T1.PT := T#0MS;
   INR_PLT4_LOCK.Error_T1.Q := FALSE;
   INR_PLT4_LOCK.Error_T1.ET := T#0MS;
   INR_PLT4_LOCK.Error_T1.STATE := B#16#0;
   INR_PLT4_LOCK.Error_T1.STIME := T#0MS;
   INR_PLT4_LOCK.Error_T1.ATIME := T#0MS;
   INR_PLT4_LOCK.Error_T2.IN := FALSE;
   INR_PLT4_LOCK.Error_T2.PT := T#0MS;
   INR_PLT4_LOCK.Error_T2.Q := FALSE;
   INR_PLT4_LOCK.Error_T2.ET := T#0MS;
   INR_PLT4_LOCK.Error_T2.STATE := B#16#0;
   INR_PLT4_LOCK.Error_T2.STIME := T#0MS;
   INR_PLT4_LOCK.Error_T2.ATIME := T#0MS;
   INR_PLT4_LOCK.CHK_Aux1 := FALSE;
   INR_PLT4_LOCK.CHK_Aux2 := FALSE;
   INR_PLT4_LOCK.Error_T1_DN := FALSE;
   INR_PLT4_LOCK.Error_T2_DN := FALSE;
   INR_PLT4_LOCK.Adv_Memo := FALSE;
   INR_PLT4_LOCK.Visu_Adv_Arr[0] := FALSE;
   INR_PLT4_LOCK.Visu_Adv_Arr[1] := FALSE;
   INR_PLT4_LOCK.Visu_Adv_Arr[2] := FALSE;
   INR_PLT4_LOCK.Visu_Adv_Arr[3] := FALSE;
   INR_PLT4_LOCK.Visu_Adv_Arr[4] := FALSE;
   INR_PLT4_LOCK.Visu_Adv_Arr[5] := FALSE;
   INR_PLT4_LOCK.Visu_Adv_Arr[6] := FALSE;
   INR_PLT4_LOCK.Visu_Adv_Arr[7] := FALSE;
   INR_PLT4_LOCK.Visu_Adv_Arr[8] := FALSE;
   INR_PLT4_LOCK.Visu_Adv_Arr[9] := FALSE;
   INR_PLT4_LOCK.Visu_Adv_Arr[10] := FALSE;
   INR_PLT4_LOCK.Visu_Adv_Arr[11] := FALSE;
   INR_PLT4_LOCK.Visu_Adv_Arr[12] := FALSE;
   INR_PLT4_LOCK.Visu_Adv_Arr[13] := FALSE;
   INR_PLT4_LOCK.Visu_Adv_Arr[14] := FALSE;
   INR_PLT4_LOCK.Visu_Adv_Arr[15] := FALSE;
   INR_PLT4_LOCK.Visu_Ret_Arr[0] := FALSE;
   INR_PLT4_LOCK.Visu_Ret_Arr[1] := FALSE;
   INR_PLT4_LOCK.Visu_Ret_Arr[2] := FALSE;
   INR_PLT4_LOCK.Visu_Ret_Arr[3] := FALSE;
   INR_PLT4_LOCK.Visu_Ret_Arr[4] := FALSE;
   INR_PLT4_LOCK.Visu_Ret_Arr[5] := FALSE;
   INR_PLT4_LOCK.Visu_Ret_Arr[6] := FALSE;
   INR_PLT4_LOCK.Visu_Ret_Arr[7] := FALSE;
   INR_PLT4_LOCK.Visu_Ret_Arr[8] := FALSE;
   INR_PLT4_LOCK.Visu_Ret_Arr[9] := FALSE;
   INR_PLT4_LOCK.Visu_Ret_Arr[10] := FALSE;
   INR_PLT4_LOCK.Visu_Ret_Arr[11] := FALSE;
   INR_PLT4_LOCK.Visu_Ret_Arr[12] := FALSE;
   INR_PLT4_LOCK.Visu_Ret_Arr[13] := FALSE;
   INR_PLT4_LOCK.Visu_Ret_Arr[14] := FALSE;
   INR_PLT4_LOCK.Visu_Ret_Arr[15] := FALSE;
   INR_PLT4_LOCK.BLK_Move_Ret := 0;
   INR_PLT4_LOCK.Enable := FALSE;
   INR_PLT4_LOCK.Adv_End := FALSE;
   INR_PLT4_LOCK.Ret_End := FALSE;
   INR_PLT5_UP_DOWN.Enable_Aux := FALSE;
   INR_PLT5_UP_DOWN.Adv_Amount := 0;
   INR_PLT5_UP_DOWN.Ret_Amount := 0;
   INR_PLT5_UP_DOWN.LS_Adv1 := FALSE;
   INR_PLT5_UP_DOWN.LS_Ret1 := FALSE;
   INR_PLT5_UP_DOWN.LS_Adv2 := FALSE;
   INR_PLT5_UP_DOWN.LS_Ret2 := FALSE;
   INR_PLT5_UP_DOWN.LS_Adv3 := FALSE;
   INR_PLT5_UP_DOWN.LS_Ret3 := FALSE;
   INR_PLT5_UP_DOWN.LS_Adv4 := FALSE;
   INR_PLT5_UP_DOWN.LS_Ret4 := FALSE;
   INR_PLT5_UP_DOWN.SOL_Adv := FALSE;
   INR_PLT5_UP_DOWN.SOL_Ret := FALSE;
   INR_PLT5_UP_DOWN.M_Ready := FALSE;
   INR_PLT5_UP_DOWN.T_CHK1 := T#0MS;
   INR_PLT5_UP_DOWN.T_CHK2 := T#0MS;
   INR_PLT5_UP_DOWN.PB_Lamp_CHK := FALSE;
   INR_PLT5_UP_DOWN.PB_Error_Rst := FALSE;
   INR_PLT5_UP_DOWN.M_FLICK := FALSE;
   INR_PLT5_UP_DOWN.M_Adv_Err := FALSE;
   INR_PLT5_UP_DOWN.M_Ret_Err := FALSE;
   INR_PLT5_UP_DOWN.LP_Adv := FALSE;
   INR_PLT5_UP_DOWN.LP_Ret := FALSE;
   INR_PLT5_UP_DOWN.Visu_Adv := W#16#0;
   INR_PLT5_UP_DOWN.Visu_Ret := W#16#0;
   INR_PLT5_UP_DOWN.Error_T1.IN := FALSE;
   INR_PLT5_UP_DOWN.Error_T1.PT := T#0MS;
   INR_PLT5_UP_DOWN.Error_T1.Q := FALSE;
   INR_PLT5_UP_DOWN.Error_T1.ET := T#0MS;
   INR_PLT5_UP_DOWN.Error_T1.STATE := B#16#0;
   INR_PLT5_UP_DOWN.Error_T1.STIME := T#0MS;
   INR_PLT5_UP_DOWN.Error_T1.ATIME := T#0MS;
   INR_PLT5_UP_DOWN.Error_T2.IN := FALSE;
   INR_PLT5_UP_DOWN.Error_T2.PT := T#0MS;
   INR_PLT5_UP_DOWN.Error_T2.Q := FALSE;
   INR_PLT5_UP_DOWN.Error_T2.ET := T#0MS;
   INR_PLT5_UP_DOWN.Error_T2.STATE := B#16#0;
   INR_PLT5_UP_DOWN.Error_T2.STIME := T#0MS;
   INR_PLT5_UP_DOWN.Error_T2.ATIME := T#0MS;
   INR_PLT5_UP_DOWN.CHK_Aux1 := FALSE;
   INR_PLT5_UP_DOWN.CHK_Aux2 := FALSE;
   INR_PLT5_UP_DOWN.Error_T1_DN := FALSE;
   INR_PLT5_UP_DOWN.Error_T2_DN := FALSE;
   INR_PLT5_UP_DOWN.Adv_Memo := FALSE;
   INR_PLT5_UP_DOWN.Visu_Adv_Arr[0] := FALSE;
   INR_PLT5_UP_DOWN.Visu_Adv_Arr[1] := FALSE;
   INR_PLT5_UP_DOWN.Visu_Adv_Arr[2] := FALSE;
   INR_PLT5_UP_DOWN.Visu_Adv_Arr[3] := FALSE;
   INR_PLT5_UP_DOWN.Visu_Adv_Arr[4] := FALSE;
   INR_PLT5_UP_DOWN.Visu_Adv_Arr[5] := FALSE;
   INR_PLT5_UP_DOWN.Visu_Adv_Arr[6] := FALSE;
   INR_PLT5_UP_DOWN.Visu_Adv_Arr[7] := FALSE;
   INR_PLT5_UP_DOWN.Visu_Adv_Arr[8] := FALSE;
   INR_PLT5_UP_DOWN.Visu_Adv_Arr[9] := FALSE;
   INR_PLT5_UP_DOWN.Visu_Adv_Arr[10] := FALSE;
   INR_PLT5_UP_DOWN.Visu_Adv_Arr[11] := FALSE;
   INR_PLT5_UP_DOWN.Visu_Adv_Arr[12] := FALSE;
   INR_PLT5_UP_DOWN.Visu_Adv_Arr[13] := FALSE;
   INR_PLT5_UP_DOWN.Visu_Adv_Arr[14] := FALSE;
   INR_PLT5_UP_DOWN.Visu_Adv_Arr[15] := FALSE;
   INR_PLT5_UP_DOWN.Visu_Ret_Arr[0] := FALSE;
   INR_PLT5_UP_DOWN.Visu_Ret_Arr[1] := FALSE;
   INR_PLT5_UP_DOWN.Visu_Ret_Arr[2] := FALSE;
   INR_PLT5_UP_DOWN.Visu_Ret_Arr[3] := FALSE;
   INR_PLT5_UP_DOWN.Visu_Ret_Arr[4] := FALSE;
   INR_PLT5_UP_DOWN.Visu_Ret_Arr[5] := FALSE;
   INR_PLT5_UP_DOWN.Visu_Ret_Arr[6] := FALSE;
   INR_PLT5_UP_DOWN.Visu_Ret_Arr[7] := FALSE;
   INR_PLT5_UP_DOWN.Visu_Ret_Arr[8] := FALSE;
   INR_PLT5_UP_DOWN.Visu_Ret_Arr[9] := FALSE;
   INR_PLT5_UP_DOWN.Visu_Ret_Arr[10] := FALSE;
   INR_PLT5_UP_DOWN.Visu_Ret_Arr[11] := FALSE;
   INR_PLT5_UP_DOWN.Visu_Ret_Arr[12] := FALSE;
   INR_PLT5_UP_DOWN.Visu_Ret_Arr[13] := FALSE;
   INR_PLT5_UP_DOWN.Visu_Ret_Arr[14] := FALSE;
   INR_PLT5_UP_DOWN.Visu_Ret_Arr[15] := FALSE;
   INR_PLT5_UP_DOWN.BLK_Move_Ret := 0;
   INR_PLT5_UP_DOWN.Enable := FALSE;
   INR_PLT5_UP_DOWN.Adv_End := FALSE;
   INR_PLT5_UP_DOWN.Ret_End := FALSE;
   INR_PLT5_LOCK.Enable_Aux := FALSE;
   INR_PLT5_LOCK.Adv_Amount := 0;
   INR_PLT5_LOCK.Ret_Amount := 0;
   INR_PLT5_LOCK.LS_Adv1 := FALSE;
   INR_PLT5_LOCK.LS_Ret1 := FALSE;
   INR_PLT5_LOCK.LS_Adv2 := FALSE;
   INR_PLT5_LOCK.LS_Ret2 := FALSE;
   INR_PLT5_LOCK.LS_Adv3 := FALSE;
   INR_PLT5_LOCK.LS_Ret3 := FALSE;
   INR_PLT5_LOCK.LS_Adv4 := FALSE;
   INR_PLT5_LOCK.LS_Ret4 := FALSE;
   INR_PLT5_LOCK.SOL_Adv := FALSE;
   INR_PLT5_LOCK.SOL_Ret := FALSE;
   INR_PLT5_LOCK.M_Ready := FALSE;
   INR_PLT5_LOCK.T_CHK1 := T#0MS;
   INR_PLT5_LOCK.T_CHK2 := T#0MS;
   INR_PLT5_LOCK.PB_Lamp_CHK := FALSE;
   INR_PLT5_LOCK.PB_Error_Rst := FALSE;
   INR_PLT5_LOCK.M_FLICK := FALSE;
   INR_PLT5_LOCK.M_Adv_Err := FALSE;
   INR_PLT5_LOCK.M_Ret_Err := FALSE;
   INR_PLT5_LOCK.LP_Adv := FALSE;
   INR_PLT5_LOCK.LP_Ret := FALSE;
   INR_PLT5_LOCK.Visu_Adv := W#16#0;
   INR_PLT5_LOCK.Visu_Ret := W#16#0;
   INR_PLT5_LOCK.Error_T1.IN := FALSE;
   INR_PLT5_LOCK.Error_T1.PT := T#0MS;
   INR_PLT5_LOCK.Error_T1.Q := FALSE;
   INR_PLT5_LOCK.Error_T1.ET := T#0MS;
   INR_PLT5_LOCK.Error_T1.STATE := B#16#0;
   INR_PLT5_LOCK.Error_T1.STIME := T#0MS;
   INR_PLT5_LOCK.Error_T1.ATIME := T#0MS;
   INR_PLT5_LOCK.Error_T2.IN := FALSE;
   INR_PLT5_LOCK.Error_T2.PT := T#0MS;
   INR_PLT5_LOCK.Error_T2.Q := FALSE;
   INR_PLT5_LOCK.Error_T2.ET := T#0MS;
   INR_PLT5_LOCK.Error_T2.STATE := B#16#0;
   INR_PLT5_LOCK.Error_T2.STIME := T#0MS;
   INR_PLT5_LOCK.Error_T2.ATIME := T#0MS;
   INR_PLT5_LOCK.CHK_Aux1 := FALSE;
   INR_PLT5_LOCK.CHK_Aux2 := FALSE;
   INR_PLT5_LOCK.Error_T1_DN := FALSE;
   INR_PLT5_LOCK.Error_T2_DN := FALSE;
   INR_PLT5_LOCK.Adv_Memo := FALSE;
   INR_PLT5_LOCK.Visu_Adv_Arr[0] := FALSE;
   INR_PLT5_LOCK.Visu_Adv_Arr[1] := FALSE;
   INR_PLT5_LOCK.Visu_Adv_Arr[2] := FALSE;
   INR_PLT5_LOCK.Visu_Adv_Arr[3] := FALSE;
   INR_PLT5_LOCK.Visu_Adv_Arr[4] := FALSE;
   INR_PLT5_LOCK.Visu_Adv_Arr[5] := FALSE;
   INR_PLT5_LOCK.Visu_Adv_Arr[6] := FALSE;
   INR_PLT5_LOCK.Visu_Adv_Arr[7] := FALSE;
   INR_PLT5_LOCK.Visu_Adv_Arr[8] := FALSE;
   INR_PLT5_LOCK.Visu_Adv_Arr[9] := FALSE;
   INR_PLT5_LOCK.Visu_Adv_Arr[10] := FALSE;
   INR_PLT5_LOCK.Visu_Adv_Arr[11] := FALSE;
   INR_PLT5_LOCK.Visu_Adv_Arr[12] := FALSE;
   INR_PLT5_LOCK.Visu_Adv_Arr[13] := FALSE;
   INR_PLT5_LOCK.Visu_Adv_Arr[14] := FALSE;
   INR_PLT5_LOCK.Visu_Adv_Arr[15] := FALSE;
   INR_PLT5_LOCK.Visu_Ret_Arr[0] := FALSE;
   INR_PLT5_LOCK.Visu_Ret_Arr[1] := FALSE;
   INR_PLT5_LOCK.Visu_Ret_Arr[2] := FALSE;
   INR_PLT5_LOCK.Visu_Ret_Arr[3] := FALSE;
   INR_PLT5_LOCK.Visu_Ret_Arr[4] := FALSE;
   INR_PLT5_LOCK.Visu_Ret_Arr[5] := FALSE;
   INR_PLT5_LOCK.Visu_Ret_Arr[6] := FALSE;
   INR_PLT5_LOCK.Visu_Ret_Arr[7] := FALSE;
   INR_PLT5_LOCK.Visu_Ret_Arr[8] := FALSE;
   INR_PLT5_LOCK.Visu_Ret_Arr[9] := FALSE;
   INR_PLT5_LOCK.Visu_Ret_Arr[10] := FALSE;
   INR_PLT5_LOCK.Visu_Ret_Arr[11] := FALSE;
   INR_PLT5_LOCK.Visu_Ret_Arr[12] := FALSE;
   INR_PLT5_LOCK.Visu_Ret_Arr[13] := FALSE;
   INR_PLT5_LOCK.Visu_Ret_Arr[14] := FALSE;
   INR_PLT5_LOCK.Visu_Ret_Arr[15] := FALSE;
   INR_PLT5_LOCK.BLK_Move_Ret := 0;
   INR_PLT5_LOCK.Enable := FALSE;
   INR_PLT5_LOCK.Adv_End := FALSE;
   INR_PLT5_LOCK.Ret_End := FALSE;
END_DATA_BLOCK

FUNCTION FC 121 : VOID
TITLE =
VERSION : 0.1

BEGIN
NETWORK
TITLE =
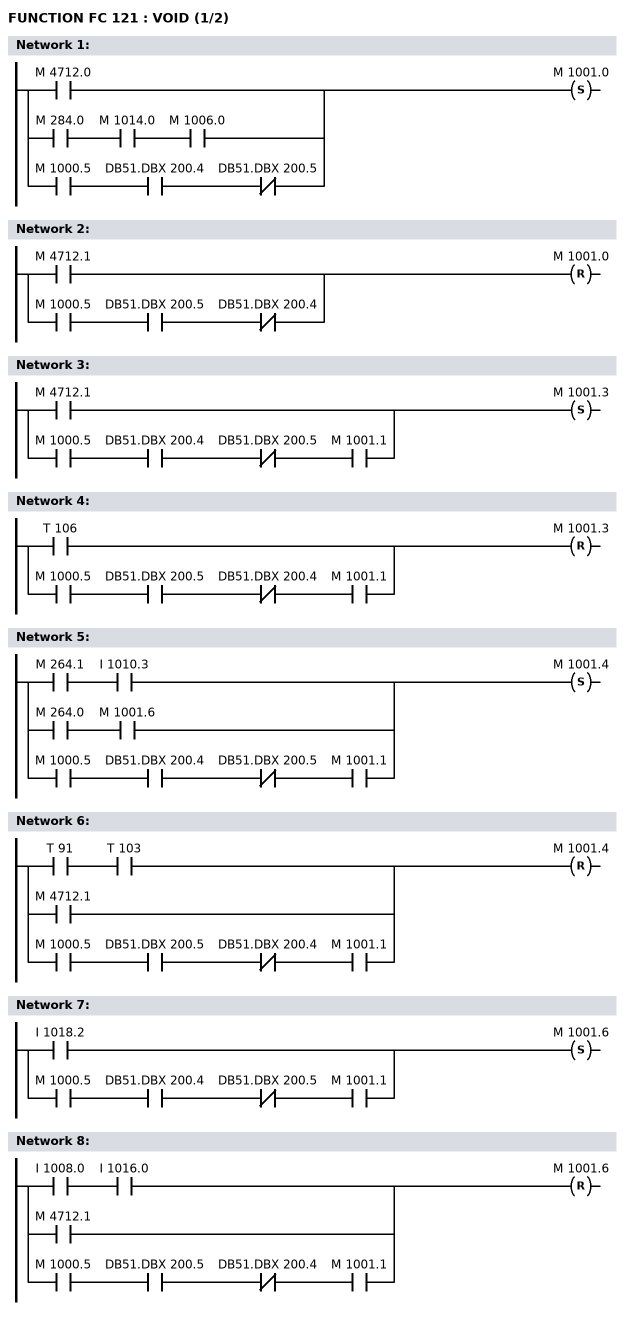

      O     M   4712.0;
      O     ;
      A     M    284.0;
      A     M   1014.0;
      A     M   1006.0;
      O     ;
      A     M   1000.5;
      A     DB51.DBX  200.4;
      AN    DB51.DBX  200.5;
      S     M   1001.0;
NETWORK
TITLE =

      O     M   4712.1;
      O     ;
      A     M   1000.5;
      A     DB51.DBX  200.5;
      AN    DB51.DBX  200.4;
      R     M   1001.0;
NETWORK
TITLE =

      O     M   4712.1;
      O     ;
      A     M   1000.5;
      A     DB51.DBX  200.4;
      AN    DB51.DBX  200.5;
      A     M   1001.1;
      S     M   1001.3;
NETWORK
TITLE =

      O     T    106;
      O     ;
      A     M   1000.5;
      A     DB51.DBX  200.5;
      AN    DB51.DBX  200.4;
      A     M   1001.1;
      R     M   1001.3;
NETWORK
TITLE =

      A     M    264.1;
      A     I   1010.3;
      O     ;
      A     M    264.0;
      A     M   1001.6;
      O     ;
      A     M   1000.5;
      A     DB51.DBX  200.4;
      AN    DB51.DBX  200.5;
      A     M   1001.1;
      S     M   1001.4;
NETWORK
TITLE =

      A     T     91;
      A     T    103;
      O     M   4712.1;
      O     ;
      A     M   1000.5;
      A     DB51.DBX  200.5;
      AN    DB51.DBX  200.4;
      A     M   1001.1;
      R     M   1001.4;
NETWORK
TITLE =

      O     I   1018.2;
      O     ;
      A     M   1000.5;
      A     DB51.DBX  200.4;
      AN    DB51.DBX  200.5;
      A     M   1001.1;
      S     M   1001.6;
NETWORK
TITLE =

      A     I   1008.0;
      A     I   1016.0;
      O     M   4712.1;
      O     ;
      A     M   1000.5;
      A     DB51.DBX  200.5;
      AN    DB51.DBX  200.4;
      A     M   1001.1;
      R     M   1001.6;
NETWORK
TITLE =
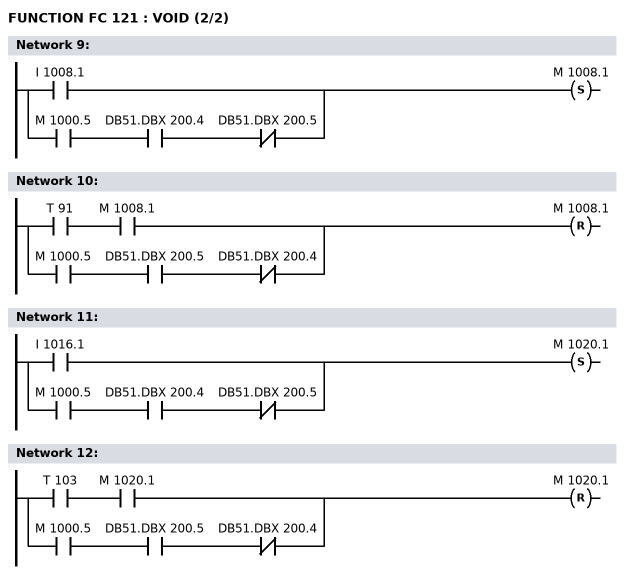

      O     I   1008.1;
      O     ;
      A     M   1000.5;
      A     DB51.DBX  200.4;
      AN    DB51.DBX  200.5;
      S     M   1008.1;
NETWORK
TITLE =

      A     T     91;
      A     M   1008.1;
      O     ;
      A     M   1000.5;
      A     DB51.DBX  200.5;
      AN    DB51.DBX  200.4;
      R     M   1008.1;
NETWORK
TITLE =

      O     I   1016.1;
      O     ;
      A     M   1000.5;
      A     DB51.DBX  200.4;
      AN    DB51.DBX  200.5;
      S     M   1020.1;
NETWORK
TITLE =

      A     T    103;
      A     M   1020.1;
      O     ;
      A     M   1000.5;
      A     DB51.DBX  200.5;
      AN    DB51.DBX  200.4;
      R     M   1020.1;
END_FUNCTION

FUNCTION_BLOCK FB 122
TITLE =
VERSION : 0.1

BEGIN
NETWORK
TITLE =
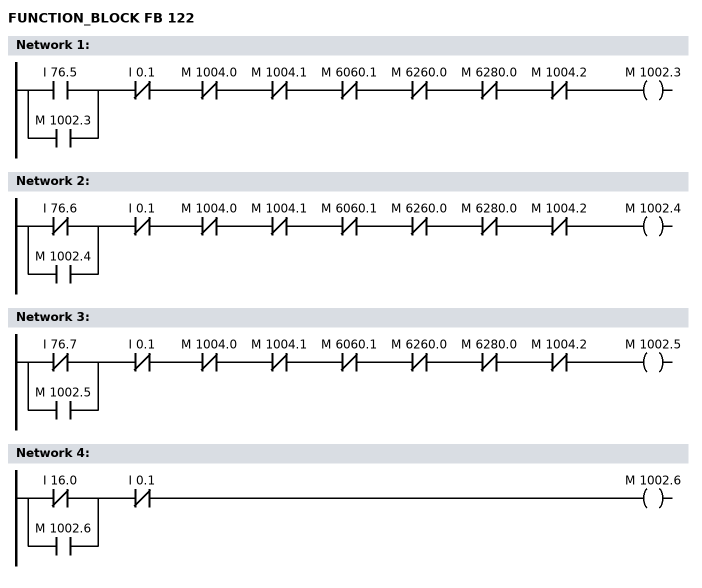

      A(    ;
      O     I     76.5;
      O     M   1002.3;
      )     ;
      AN    I      0.1;
      AN    M   1004.0;
      AN    M   1004.1;
      AN    M   6060.1;
      AN    M   6260.0;
      AN    M   6280.0;
      AN    M   1004.2;
      =     M   1002.3;
NETWORK
TITLE =

      A(    ;
      ON    I     76.6;
      O     M   1002.4;
      )     ;
      AN    I      0.1;
      AN    M   1004.0;
      AN    M   1004.1;
      AN    M   6060.1;
      AN    M   6260.0;
      AN    M   6280.0;
      AN    M   1004.2;
      =     M   1002.4;
NETWORK
TITLE =

      A(    ;
      ON    I     76.7;
      O     M   1002.5;
      )     ;
      AN    I      0.1;
      AN    M   1004.0;
      AN    M   1004.1;
      AN    M   6060.1;
      AN    M   6260.0;
      AN    M   6280.0;
      AN    M   1004.2;
      =     M   1002.5;
NETWORK
TITLE =

      A(    ;
      ON    I     16.0;
      O     M   1002.6;
      )     ;
      AN    I      0.1;
      =     M   1002.6;
NETWORK
TITLE =

